LIN {X 0,Y 688.052,Z 1286.33,A -85,B 0,C 180,E1 33039.113,E2 33039.113} C_VEL
LIN {X 0,Y 687.976,Z 1293.841,A -85,B 0,C 180,E1 33037.347,E2 33037.347} C_VEL
LIN {X 0,Y 687.922,Z 1299.397,A -85,B 0,C 180,E1 33035.671,E2 33035.671} C_VEL
LIN {X 0,Y 687.911,Z 1303.97,A -85,B 0,C 180,E1 33033.749,E2 33033.749} C_VEL
LIN {X 0,Y 687.912,Z 1306.541,A -85,B 0,C 180,E1 33031.915,E2 33031.915} C_VEL
LIN {X 0,Y 687.913,Z 1307.484,A -85,B 0,C 180,E1 33030.082,E2 33030.082} C_VEL
LIN {X 0,Y 687.914,Z 1306.622,A -85,B 0,C 180,E1 33028.166,E2 33028.166} C_VEL
LIN {X 0,Y 687.914,Z 1304.122,A -85,B 0,C 180,E1 33026.332,E2 33026.332} C_VEL
LIN {X 0,Y 687.924,Z 1299.644,A -85,B 0,C 180,E1 33024.41,E2 33024.41} C_VEL
LIN {X 0,Y 687.974,Z 1294.146,A -85,B 0,C 180,E1 33022.735,E2 33022.735} C_VEL
LIN {X 0,Y 688.047,Z 1286.725,A -85,B 0,C 180,E1 33020.969,E2 33020.969} C_VEL
LIN {X 0,Y 688.172,Z 1277.229,A -85,B 0,C 180,E1 33019.176,E2 33019.176} C_VEL
LIN {X 0,Y 688.352,Z 1267.627,A -85,B 0,C 180,E1 33017.67,E2 33017.67} C_VEL
LIN {X 0,Y 688.626,Z 1255.593,A -85,B 0,C 180,E1 33016.052,E2 33016.052} C_VEL
LIN {X 0,Y 688.958,Z 1242.007,A -85,B 0,C 180,E1 33014.509,E2 33014.509} C_VEL
LIN {X 0,Y 689.355,Z 1227.995,A -85,B 0,C 180,E1 33013.136,E2 33013.136} C_VEL
LIN {X 0,Y 689.893,Z 1210.597,A -85,B 0,C 180,E1 33011.668,E2 33011.668} C_VEL
LIN {X 0,Y 690.479,Z 1192.469,A -85,B 0,C 180,E1 33010.368,E2 33010.368} C_VEL
LIN {X 0,Y 691.054,Z 1173.913,A -85,B 0,C 180,E1 33009.237,E2 33009.237} C_VEL
LIN {X 0,Y 691.686,Z 1153.527,A -85,B 0,C 180,E1 33008.19,E2 33008.19} C_VEL
LIN {X 0,Y 692.271,Z 1132.946,A -85,B 0,C 180,E1 33007.315,E2 33007.315} C_VEL
LIN {X 0,Y 692.788,Z 1111.812,A -85,B 0,C 180,E1 33006.587,E2 33006.587} C_VEL
LIN {X 0,Y 693.277,Z 1089.541,A -85,B 0,C 180,E1 33005.995,E2 33005.995} C_VEL
LIN {X 0,Y 693.611,Z 1067.293,A -85,B 0,C 180,E1 33005.565,E2 33005.565} C_VEL
LIN {X 0,Y 693.882,Z 1034.911,A -85,B 0,C 180,E1 33005.171,E2 33005.171} C_VEL
LIN {X 0,Y 694.12,Z 1007.188,A -85,B 0,C 180,E1 33004.852,E2 33004.852} C_VEL
LIN {X 0,Y 696.375,Z 998.353,A -85,B 0,C 180,E1 33004.529,E2 33004.529} C_VEL
LIN {X 0,Y 699.809,Z 987.003,A -85,B 0,C 180,E1 33004.278,E2 33004.278} C_VEL
LIN {X 0,Y 700.607,Z 984.081,A -85,B 0,C 180,E1 33004.196,E2 33004.196} C_VEL
LIN {X 0,Y 703.226,Z 974.14,A -85,B 0,C 180,E1 33003.891,E2 33003.891} C_VEL
LIN {X 0,Y 707.415,Z 958.39,A -85,B 0,C 180,E1 33003.611,E2 33003.611} C_VEL
LIN {X 0,Y 711.232,Z 939.749,A -85,B 0,C 180,E1 33003.422,E2 33003.422} C_VEL
LIN {X 0,Y 713.381,Z 919.951,A -85,B 0,C 180,E1 33003.244,E2 33003.244} C_VEL
LIN {X 0,Y 716.131,Z 876.116,A -85,B 0,C 180,E1 33002.811,E2 33002.811} C_VEL
LIN {X 0,Y 717.751,Z 866.34,A -85,B 0,C 180,E1 33002.56,E2 33002.56} C_VEL
LIN {X 0,Y 720.347,Z 841.246,A -85,B 0,C 180,E1 33002.165,E2 33002.165} C_VEL
LIN {X 0,Y 724.376,Z 790.008,A -85,B 0,C 180,E1 33001.568,E2 33001.568} C_VEL
LIN {X 0,Y 725.039,Z 781.425,A -85,B 0,C 180,E1 33001.471,E2 33001.471} C_VEL
LIN {X 0,Y 727.199,Z 793.678,A -85,B 0,C 180,E1 33001.159,E2 33001.159} C_VEL
LIN {X 0,Y 730.142,Z 804.778,A -85,B 0,C 180,E1 33000.743,E2 33000.743} C_VEL
LIN {X 0,Y 733.96,Z 814.871,A -85,B 0,C 180,E1 33000.215,E2 33000.215} C_VEL
LIN {X 0,Y 738.534,Z 823.545,A -85,B 0,C 180,E1 32999.601,E2 32999.601} C_VEL
LIN {X 0,Y 740.672,Z 827.583,A -85,B 0,C 180,E1 32999.211,E2 32999.211} C_VEL
LIN {X 0,Y 741.307,Z 830.76,A -85,B 0,C 180,E1 32998.777,E2 32998.777} C_VEL
LIN {X 0,Y 740.425,Z 833.197,A -85,B 0,C 180,E1 32998.296,E2 32998.296} C_VEL
LIN {X 0,Y 738.218,Z 834.451,A -85,B 0,C 180,E1 32997.838,E2 32997.838} C_VEL
LIN {X 0,Y 734.644,Z 834.531,A -85,B 0,C 180,E1 32997.385,E2 32997.385} C_VEL
LIN {X 0,Y 730.605,Z 833.461,A -85,B 0,C 180,E1 32997.029,E2 32997.029} C_VEL
LIN {X 0,Y 722.325,Z 829.141,A -85,B 0,C 180,E1 32996.443,E2 32996.443} C_VEL
LIN {X 0,Y 715.279,Z 823.545,A -85,B 0,C 180,E1 32995.849,E2 32995.849} C_VEL
LIN {X 0,Y 709.495,Z 816.874,A -85,B 0,C 180,E1 32995.248,E2 32995.248} C_VEL
LIN {X 0,Y 704.432,Z 808.219,A -85,B 0,C 180,E1 32994.563,E2 32994.563} C_VEL
LIN {X 0,Y 700.551,Z 797.694,A -85,B 0,C 180,E1 32993.817,E2 32993.817} C_VEL
LIN {X 0,Y 697.983,Z 785.051,A -85,B 0,C 180,E1 32993.01,E2 32993.01} C_VEL
LIN {X 0,Y 696.676,Z 766.868,A -85,B 0,C 180,E1 32991.949,E2 32991.949} C_VEL
LIN {X 0,Y 698.246,Z 704.476,A -85,B 0,C 180,E1 32988.524,E2 32988.524} C_VEL
LIN {X 0,Y 699.163,Z 671.327,A -85,B 0,C 180,E1 32986.649,E2 32986.649} C_VEL
LIN {X 0,Y 689.472,Z 649.922,A -85,B 0,C 180,E1 32984.698,E2 32984.698} C_VEL
LIN {X 0,Y 688.454,Z 646.906,A -85,B 0,C 180,E1 32984.431,E2 32984.431} C_VEL
LIN {X 0,Y 688.446,Z 646.914,A -85,B 0,C 180,E1 32981.458,E2 32981.458} C_VEL
LIN {X 0,Y 688.453,Z 646.914,A -85,B 0,C 180,E1 32978.479,E2 32978.479} C_VEL
LIN {X 0,Y 688.465,Z 646.915,A -85,B 0,C 180,E1 32975.435,E2 32975.435} C_VEL
LIN {X 0,Y 688.476,Z 647.124,A -85,B 0,C 180,E1 32972.456,E2 32972.456} C_VEL
LIN {X 0,Y 693.195,Z 663.428,A -85,B 0,C 180,E1 32970.946,E2 32970.946} C_VEL
LIN {X 0,Y 692.593,Z 691.38,A -85,B 0,C 180,E1 32968.687,E2 32968.687} C_VEL
LIN {X 0,Y 692.429,Z 700.611,A -85,B 0,C 180,E1 32967.953,E2 32967.953} C_VEL
LIN {X 0,Y 695.311,Z 714.317,A -85,B 0,C 180,E1 32967.669,E2 32967.669} C_VEL
LIN {X 0,Y 693.776,Z 994.51,A -85,B 0,C 180,E1 32964.567,E2 32964.567} C_VEL
LIN {X 0,Y 693.492,Z 1016.407,A -85,B 0,C 180,E1 32964.232,E2 32964.232} C_VEL
LIN {X 0,Y 693.064,Z 1038.792,A -85,B 0,C 180,E1 32963.733,E2 32963.733} C_VEL
LIN {X 0,Y 692.622,Z 1059.513,A -85,B 0,C 180,E1 32963.121,E2 32963.121} C_VEL
LIN {X 0,Y 692.072,Z 1079.43,A -85,B 0,C 180,E1 32962.383,E2 32962.383} C_VEL
LIN {X 0,Y 691.52,Z 1098.933,A -85,B 0,C 180,E1 32961.503,E2 32961.503} C_VEL
LIN {X 0,Y 690.941,Z 1117.723,A -85,B 0,C 180,E1 32960.5,E2 32960.5} C_VEL
LIN {X 0,Y 690.349,Z 1136.287,A -85,B 0,C 180,E1 32959.331,E2 32959.331} C_VEL
LIN {X 0,Y 689.813,Z 1153.31,A -85,B 0,C 180,E1 32958.071,E2 32958.071} C_VEL
LIN {X 0,Y 689.325,Z 1169.406,A -85,B 0,C 180,E1 32956.691,E2 32956.691} C_VEL
LIN {X 0,Y 688.911,Z 1184.069,A -85,B 0,C 180,E1 32955.231,E2 32955.231} C_VEL
LIN {X 0,Y 688.574,Z 1197.285,A -85,B 0,C 180,E1 32953.692,E2 32953.692} C_VEL
LIN {X 0,Y 688.318,Z 1209.092,A -85,B 0,C 180,E1 32952.075,E2 32952.075} C_VEL
LIN {X 0,Y 688.136,Z 1219.976,A -85,B 0,C 180,E1 32950.296,E2 32950.296} C_VEL
LIN {X 0,Y 688.015,Z 1228.491,A -85,B 0,C 180,E1 32948.609,E2 32948.609} C_VEL
LIN {X 0,Y 687.957,Z 1235.51,A -85,B 0,C 180,E1 32946.845,E2 32946.845} C_VEL
LIN {X 0,Y 687.914,Z 1241.082,A -85,B 0,C 180,E1 32945.003,E2 32945.003} C_VEL
LIN {X 0,Y 687.904,Z 1244.799,A -85,B 0,C 180,E1 32943.25,E2 32943.25} C_VEL
LIN {X 0,Y 687.909,Z 1246.913,A -85,B 0,C 180,E1 32941.416,E2 32941.416} C_VEL
LIN {X 0,Y 687.917,Z 1247.386,A -85,B 0,C 180,E1 32939.5,E2 32939.5} C_VEL
LIN {X 0,Y 687.906,Z 1246.182,A -85,B 0,C 180,E1 32937.667,E2 32937.667} C_VEL
LIN {X 0,Y 687.903,Z 1243.392,A -85,B 0,C 180,E1 32935.916,E2 32935.916} C_VEL
LIN {X 0,Y 687.927,Z 1238.788,A -85,B 0,C 180,E1 32934.077,E2 32934.077} C_VEL
LIN {X 0,Y 687.972,Z 1232.769,A -85,B 0,C 180,E1 32932.316,E2 32932.316} C_VEL
LIN {X 0,Y 688.058,Z 1224.885,A -85,B 0,C 180,E1 32930.548,E2 32930.548} C_VEL
LIN {X 0,Y 688.219,Z 1215.089,A -85,B 0,C 180,E1 32928.774,E2 32928.774} C_VEL
LIN {X 0,Y 688.427,Z 1203.628,A -85,B 0,C 180,E1 32927.054,E2 32927.054} C_VEL
LIN {X 0,Y 688.733,Z 1191.01,A -85,B 0,C 180,E1 32925.454,E2 32925.454} C_VEL
LIN {X 0,Y 689.115,Z 1176.622,A -85,B 0,C 180,E1 32923.911,E2 32923.911} C_VEL
LIN {X 0,Y 689.566,Z 1161.193,A -85,B 0,C 180,E1 32922.489,E2 32922.489} C_VEL
LIN {X 0,Y 690.092,Z 1144.286,A -85,B 0,C 180,E1 32921.149,E2 32921.149} C_VEL
LIN {X 0,Y 690.664,Z 1126.45,A -85,B 0,C 180,E1 32919.933,E2 32919.933} C_VEL
LIN {X 0,Y 691.261,Z 1107.52,A -85,B 0,C 180,E1 32918.845,E2 32918.845} C_VEL
LIN {X 0,Y 691.847,Z 1087.678,A -85,B 0,C 180,E1 32917.882,E2 32917.882} C_VEL
LIN {X 0,Y 692.178,Z 1075.526,A -85,B 0,C 180,E1 32917.373,E2 32917.373} C_VEL
LIN {X 0,Y 691.49,Z 1068.665,A -85,B 0,C 180,E1 32917.076,E2 32917.076} C_VEL
LIN {X 0,Y 686.397,Z 1051.614,A -85,B 0,C 180,E1 32916.295,E2 32916.295} C_VEL
LIN {X 0,Y 685.615,Z 1044.451,A -85,B 0,C 180,E1 32916.058,E2 32916.058} C_VEL
LIN {X 0,Y 686.063,Z 1022.443,A -85,B 0,C 180,E1 32915.52,E2 32915.52} C_VEL
LIN {X 0,Y 686.423,Z 1000.492,A -85,B 0,C 180,E1 32915.146,E2 32915.146} C_VEL
LIN {X 0,Y 688.095,Z 732.537,A -85,B 0,C 180,E1 32912.14,E2 32912.14} C_VEL
LIN {X 0,Y 687.988,Z 713.74,A -85,B 0,C 180,E1 32911.919,E2 32911.919} C_VEL
LIN {X 0,Y 684.931,Z 700.129,A -85,B 0,C 180,E1 32911.605,E2 32911.605} C_VEL
LIN {X 0,Y 685.853,Z 667.016,A -85,B 0,C 180,E1 32908.881,E2 32908.881} C_VEL
LIN {X 0,Y 685.402,Z 664.065,A -85,B 0,C 180,E1 32908.614,E2 32908.614} C_VEL
LIN {X 0,Y 680.514,Z 647.904,A -85,B 0,C 180,E1 32906.992,E2 32906.992} C_VEL
LIN {X 0,Y 680.521,Z 647.902,A -85,B 0,C 180,E1 32903.9,E2 32903.9} C_VEL
LIN {X 0,Y 680.516,Z 647.9,A -85,B 0,C 180,E1 32900.816,E2 32900.816} C_VEL
LIN {X 0,Y 680.522,Z 647.897,A -85,B 0,C 180,E1 32897.777,E2 32897.777} C_VEL
LIN {X 0,Y 680.52,Z 647.9,A -85,B 0,C 180,E1 32894.615,E2 32894.615} C_VEL
LIN {X 0,Y 680.53,Z 647.902,A -85,B 0,C 180,E1 32891.503,E2 32891.503} C_VEL
LIN {X 0,Y 680.525,Z 647.898,A -85,B 0,C 180,E1 32888.427,E2 32888.427} C_VEL
LIN {X 0,Y 680.52,Z 647.896,A -85,B 0,C 180,E1 32885.271,E2 32885.271} C_VEL
LIN {X 0,Y 680.519,Z 647.898,A -85,B 0,C 180,E1 32882.134,E2 32882.134} C_VEL
LIN {X 0,Y 680.531,Z 647.902,A -85,B 0,C 180,E1 32879.046,E2 32879.046} C_VEL
LIN {X 0,Y 680.521,Z 647.896,A -85,B 0,C 180,E1 32875.945,E2 32875.945} C_VEL
LIN {X 0,Y 680.524,Z 647.895,A -85,B 0,C 180,E1 32872.824,E2 32872.824} C_VEL
LIN {X 0,Y 680.52,Z 647.897,A -85,B 0,C 180,E1 32869.663,E2 32869.663} C_VEL
LIN {X 0,Y 680.525,Z 647.902,A -85,B 0,C 180,E1 32866.562,E2 32866.562} C_VEL
LIN {X 0,Y 680.523,Z 647.894,A -85,B 0,C 180,E1 32863.511,E2 32863.511} C_VEL
LIN {X 0,Y 680.521,Z 647.895,A -85,B 0,C 180,E1 32860.327,E2 32860.327} C_VEL
LIN {X 0,Y 680.521,Z 647.898,A -85,B 0,C 180,E1 32857.175,E2 32857.175} C_VEL
LIN {X 0,Y 680.522,Z 647.901,A -85,B 0,C 180,E1 32854.13,E2 32854.13} C_VEL
LIN {X 0,Y 680.524,Z 647.896,A -85,B 0,C 180,E1 32851.011,E2 32851.011} C_VEL
LIN {X 0,Y 680.523,Z 647.895,A -85,B 0,C 180,E1 32847.896,E2 32847.896} C_VEL
LIN {X 0,Y 680.522,Z 647.899,A -85,B 0,C 180,E1 32844.775,E2 32844.775} C_VEL
LIN {X 0,Y 680.525,Z 647.899,A -85,B 0,C 180,E1 32841.722,E2 32841.722} C_VEL
LIN {X 0,Y 680.522,Z 647.894,A -85,B 0,C 180,E1 32838.561,E2 32838.561} C_VEL
LIN {X 0,Y 680.524,Z 647.893,A -85,B 0,C 180,E1 32835.363,E2 32835.363} C_VEL
LIN {X 0,Y 680.52,Z 647.898,A -85,B 0,C 180,E1 32832.197,E2 32832.197} C_VEL
LIN {X 0,Y 680.524,Z 647.903,A -85,B 0,C 180,E1 32829.083,E2 32829.083} C_VEL
LIN {X 0,Y 680.524,Z 647.897,A -85,B 0,C 180,E1 32826.051,E2 32826.051} C_VEL
LIN {X 0,Y 680.526,Z 647.894,A -85,B 0,C 180,E1 32822.906,E2 32822.906} C_VEL
LIN {X 0,Y 680.522,Z 647.898,A -85,B 0,C 180,E1 32819.739,E2 32819.739} C_VEL
LIN {X 0,Y 680.524,Z 647.899,A -85,B 0,C 180,E1 32816.668,E2 32816.668} C_VEL
LIN {X 0,Y 680.521,Z 647.894,A -85,B 0,C 180,E1 32813.589,E2 32813.589} C_VEL
LIN {X 0,Y 680.528,Z 647.895,A -85,B 0,C 180,E1 32810.478,E2 32810.478} C_VEL
LIN {X 0,Y 680.518,Z 647.901,A -85,B 0,C 180,E1 32807.278,E2 32807.278} C_VEL
LIN {X 0,Y 680.525,Z 647.902,A -85,B 0,C 180,E1 32804.194,E2 32804.194} C_VEL
LIN {X 0,Y 680.516,Z 647.983,A -85,B 0,C 180,E1 32801.533,E2 32801.533} C_VEL
LIN {X 0,Y 687.339,Z 668.46,A -85,B 0,C 180,E1 32799.641,E2 32799.641} C_VEL
LIN {X 0,Y 686.324,Z 710.17,A -85,B 0,C 180,E1 32796.678,E2 32796.678} C_VEL
LIN {X 0,Y 685.036,Z 755.985,A -85,B 0,C 180,E1 32793.486,E2 32793.486} C_VEL
LIN {X 0,Y 683.854,Z 801.811,A -85,B 0,C 180,E1 32790.343,E2 32790.343} C_VEL
LIN {X 0,Y 682.807,Z 848.451,A -85,B 0,C 180,E1 32787.187,E2 32787.187} C_VEL
LIN {X 0,Y 681.979,Z 893.847,A -85,B 0,C 180,E1 32784.163,E2 32784.163} C_VEL
LIN {X 0,Y 682.461,Z 901.344,A -85,B 0,C 180,E1 32784.057,E2 32784.057} C_VEL
LIN {X 0,Y 681.831,Z 1024.236,A -85,B 0,C 180,E1 32782.694,E2 32782.694} C_VEL
LIN {X 0,Y 681.705,Z 1043.086,A -85,B 0,C 180,E1 32782.409,E2 32782.409} C_VEL
LIN {X 0,Y 681.562,Z 1057.156,A -85,B 0,C 180,E1 32782.059,E2 32782.059} C_VEL
LIN {X 0,Y 681.374,Z 1070.311,A -85,B 0,C 180,E1 32781.613,E2 32781.613} C_VEL
LIN {X 0,Y 681.169,Z 1082.604,A -85,B 0,C 180,E1 32781.078,E2 32781.078} C_VEL
LIN {X 0,Y 680.956,Z 1094.166,A -85,B 0,C 180,E1 32780.455,E2 32780.455} C_VEL
LIN {X 0,Y 680.77,Z 1105.02,A -85,B 0,C 180,E1 32779.744,E2 32779.744} C_VEL
LIN {X 0,Y 680.576,Z 1115.127,A -85,B 0,C 180,E1 32778.947,E2 32778.947} C_VEL
LIN {X 0,Y 680.397,Z 1124.558,A -85,B 0,C 180,E1 32778.052,E2 32778.052} C_VEL
LIN {X 0,Y 680.233,Z 1133.602,A -85,B 0,C 180,E1 32777.009,E2 32777.009} C_VEL
LIN {X 0,Y 680.099,Z 1142.811,A -85,B 0,C 180,E1 32775.645,E2 32775.645} C_VEL
LIN {X 0,Y 680.029,Z 1148.744,A -85,B 0,C 180,E1 32774.475,E2 32774.475} C_VEL
LIN {X 0,Y 679.997,Z 1153.042,A -85,B 0,C 180,E1 32773.348,E2 32773.348} C_VEL
LIN {X 0,Y 679.98,Z 1156.037,A -85,B 0,C 180,E1 32772.225,E2 32772.225} C_VEL
LIN {X 0,Y 679.976,Z 1157.82,A -85,B 0,C 180,E1 32771.107,E2 32771.107} C_VEL
LIN {X 0,Y 679.976,Z 1158.446,A -85,B 0,C 180,E1 32769.992,E2 32769.992} C_VEL
LIN {X 0,Y 679.98,Z 1157.896,A -85,B 0,C 180,E1 32768.841,E2 32768.841} C_VEL
LIN {X 0,Y 679.989,Z 1156.299,A -85,B 0,C 180,E1 32767.775,E2 32767.775} C_VEL
LIN {X 0,Y 680.009,Z 1153.501,A -85,B 0,C 180,E1 32766.671,E2 32766.671} C_VEL
LIN {X 0,Y 680.043,Z 1149.483,A -85,B 0,C 180,E1 32765.569,E2 32765.569} C_VEL
LIN {X 0,Y 680.109,Z 1144.147,A -85,B 0,C 180,E1 32764.469,E2 32764.469} C_VEL
LIN {X 0,Y 680.215,Z 1137.348,A -85,B 0,C 180,E1 32763.371,E2 32763.371} C_VEL
LIN {X 0,Y 680.395,Z 1128.078,A -85,B 0,C 180,E1 32762.185,E2 32762.185} C_VEL
LIN {X 0,Y 680.619,Z 1117.182,A -85,B 0,C 180,E1 32761.094,E2 32761.094} C_VEL
LIN {X 0,Y 680.839,Z 1106.279,A -85,B 0,C 180,E1 32760.21,E2 32760.21} C_VEL
LIN {X 0,Y 681.041,Z 1095.617,A -85,B 0,C 180,E1 32759.495,E2 32759.495} C_VEL
LIN {X 0,Y 681.246,Z 1084.216,A -85,B 0,C 180,E1 32758.865,E2 32758.865} C_VEL
LIN {X 0,Y 681.48,Z 1071.988,A -85,B 0,C 180,E1 32758.318,E2 32758.318} C_VEL
LIN {X 0,Y 681.666,Z 1058.753,A -85,B 0,C 180,E1 32757.856,E2 32757.856} C_VEL
LIN {X 0,Y 681.814,Z 1044.156,A -85,B 0,C 180,E1 32757.484,E2 32757.484} C_VEL
LIN {X 0,Y 681.926,Z 1026.393,A -85,B 0,C 180,E1 32757.206,E2 32757.206} C_VEL
LIN {X 0,Y 682.494,Z 951.65,A -85,B 0,C 180,E1 32756.322,E2 32756.322} C_VEL
LIN {X 0,Y 682.806,Z 896.544,A -85,B 0,C 180,E1 32755.66,E2 32755.66} C_VEL
LIN {X 0,Y 682.86,Z 890.86,A -85,B 0,C 180,E1 32755.296,E2 32755.296} C_VEL
LIN {X 0,Y 684.314,Z 844.923,A -85,B 0,C 180,E1 32752.106,E2 32752.106} C_VEL
LIN {X 0,Y 686.061,Z 799.923,A -85,B 0,C 180,E1 32748.908,E2 32748.908} C_VEL
LIN {X 0,Y 688.301,Z 755.929,A -85,B 0,C 180,E1 32745.702,E2 32745.702} C_VEL
LIN {X 0,Y 690.915,Z 714.185,A -85,B 0,C 180,E1 32742.568,E2 32742.568} C_VEL
LIN {X 0,Y 692.798,Z 677.036,A -85,B 0,C 180,E1 32739.601,E2 32739.601} C_VEL
LIN {X 0,Y 687.372,Z 663.531,A -85,B 0,C 180,E1 32737.908,E2 32737.908} C_VEL
LIN {X 0,Y 683.533,Z 655.104,A -85,B 0,C 180,E1 32736.725,E2 32736.725} C_VEL
LIN {X 0,Y 682.014,Z 651.668,A -85,B 0,C 180,E1 32736.223,E2 32736.223} C_VEL
LIN {X 0,Y 680.706,Z 648.913,A -85,B 0,C 180,E1 32735.804,E2 32735.804} C_VEL
LIN {X 0,Y 680.52,Z 647.9,A -85,B 0,C 180,E1 32735.671,E2 32735.671} C_VEL
LIN {X 0,Y 680.52,Z 647.902,A -85,B 0,C 180,E1 32732.525,E2 32732.525} C_VEL
LIN {X 0,Y 680.526,Z 647.898,A -85,B 0,C 180,E1 32729.346,E2 32729.346} C_VEL
LIN {X 0,Y 680.522,Z 647.904,A -85,B 0,C 180,E1 32726.161,E2 32726.161} C_VEL
LIN {X 0,Y 680.524,Z 647.898,A -85,B 0,C 180,E1 32723.06,E2 32723.06} C_VEL
LIN {X 0,Y 680.527,Z 647.901,A -85,B 0,C 180,E1 32719.943,E2 32719.943} C_VEL
LIN {X 0,Y 680.523,Z 647.9,A -85,B 0,C 180,E1 32716.781,E2 32716.781} C_VEL
LIN {X 0,Y 680.537,Z 648.001,A -85,B 0,C 180,E1 32715.741,E2 32715.741} C_VEL
LIN {X 0,Y 681.774,Z 651.333,A -85,B 0,C 180,E1 32715.372,E2 32715.372} C_VEL
LIN {X 0,Y 682.888,Z 653.487,A -85,B 0,C 180,E1 32715.11,E2 32715.11} C_VEL
LIN {X 0,Y 687.786,Z 664.015,A -85,B 0,C 180,E1 32713.976,E2 32713.976} C_VEL
LIN {X 0,Y 691.216,Z 672.497,A -85,B 0,C 180,E1 32713.172,E2 32713.172} C_VEL
LIN {X 0,Y 688.619,Z 719.746,A -85,B 0,C 180,E1 32710.523,E2 32710.523} C_VEL
LIN {X 0,Y 687.369,Z 766.196,A -85,B 0,C 180,E1 32708.026,E2 32708.026} C_VEL
LIN {X 0,Y 688.944,Z 785.514,A -85,B 0,C 180,E1 32706.929,E2 32706.929} C_VEL
LIN {X 0,Y 692.056,Z 799.714,A -85,B 0,C 180,E1 32706.062,E2 32706.062} C_VEL
LIN {X 0,Y 696.525,Z 811.165,A -85,B 0,C 180,E1 32705.303,E2 32705.303} C_VEL
LIN {X 0,Y 702.239,Z 820.654,A -85,B 0,C 180,E1 32704.614,E2 32704.614} C_VEL
LIN {X 0,Y 709.083,Z 828.478,A -85,B 0,C 180,E1 32703.988,E2 32703.988} C_VEL
LIN {X 0,Y 717.318,Z 835.074,A -85,B 0,C 180,E1 32703.388,E2 32703.388} C_VEL
LIN {X 0,Y 726.337,Z 840.033,A -85,B 0,C 180,E1 32702.844,E2 32702.844} C_VEL
LIN {X 0,Y 731.268,Z 841.551,A -85,B 0,C 180,E1 32702.472,E2 32702.472} C_VEL
LIN {X 0,Y 735.317,Z 841.711,A -85,B 0,C 180,E1 32702.026,E2 32702.026} C_VEL
LIN {X 0,Y 738.021,Z 840.588,A -85,B 0,C 180,E1 32701.549,E2 32701.549} C_VEL
LIN {X 0,Y 739.249,Z 838.373,A -85,B 0,C 180,E1 32701.068,E2 32701.068} C_VEL
LIN {X 0,Y 738.904,Z 835.208,A -85,B 0,C 180,E1 32700.603,E2 32700.603} C_VEL
LIN {X 0,Y 737.005,Z 831.347,A -85,B 0,C 180,E1 32700.197,E2 32700.197} C_VEL
LIN {X 0,Y 732.153,Z 822.678,A -85,B 0,C 180,E1 32699.537,E2 32699.537} C_VEL
LIN {X 0,Y 728.061,Z 812.657,A -85,B 0,C 180,E1 32698.964,E2 32698.964} C_VEL
LIN {X 0,Y 726.84,Z 809.083,A -85,B 0,C 180,E1 32698.789,E2 32698.789} C_VEL
LIN {X 0,Y 723.154,Z 852.196,A -85,B 0,C 180,E1 32698.253,E2 32698.253} C_VEL
LIN {X 0,Y 720.83,Z 872.102,A -85,B 0,C 180,E1 32697.907,E2 32697.907} C_VEL
LIN {X 0,Y 719.496,Z 880.295,A -85,B 0,C 180,E1 32697.706,E2 32697.706} C_VEL
LIN {X 0,Y 717.196,Z 912.709,A -85,B 0,C 180,E1 32697.417,E2 32697.417} C_VEL
LIN {X 0,Y 713.888,Z 932.091,A -85,B 0,C 180,E1 32697.277,E2 32697.277} C_VEL
LIN {X 0,Y 708.832,Z 950.724,A -85,B 0,C 180,E1 32697.129,E2 32697.129} C_VEL
LIN {X 0,Y 703.102,Z 967.543,A -85,B 0,C 180,E1 32696.885,E2 32696.885} C_VEL
LIN {X 0,Y 698.713,Z 980.481,A -85,B 0,C 180,E1 32696.567,E2 32696.567} C_VEL
LIN {X 0,Y 696.39,Z 988.262,A -85,B 0,C 180,E1 32696.311,E2 32696.311} C_VEL
LIN {X 0,Y 691.992,Z 1000.207,A -85,B 0,C 180,E1 32696.004,E2 32696.004} C_VEL
LIN {X 0,Y 686.96,Z 1018.232,A -85,B 0,C 180,E1 32695.334,E2 32695.334} C_VEL
LIN {X 0,Y 686.704,Z 1020.499,A -85,B 0,C 180,E1 32695.269,E2 32695.269} C_VEL
LIN {X 0,Y 686.367,Z 1064.962,A -85,B 0,C 180,E1 32694.747,E2 32694.747} C_VEL
LIN {X 0,Y 685.968,Z 1087.624,A -85,B 0,C 180,E1 32694.321,E2 32694.321} C_VEL
LIN {X 0,Y 685.459,Z 1109.858,A -85,B 0,C 180,E1 32693.74,E2 32693.74} C_VEL
LIN {X 0,Y 684.902,Z 1130.772,A -85,B 0,C 180,E1 32693.031,E2 32693.031} C_VEL
LIN {X 0,Y 684.264,Z 1150.713,A -85,B 0,C 180,E1 32692.196,E2 32692.196} C_VEL
LIN {X 0,Y 683.586,Z 1170.799,A -85,B 0,C 180,E1 32691.178,E2 32691.178} C_VEL
LIN {X 0,Y 682.88,Z 1190.505,A -85,B 0,C 180,E1 32689.991,E2 32689.991} C_VEL
LIN {X 0,Y 682.27,Z 1207.173,A -85,B 0,C 180,E1 32688.808,E2 32688.808} C_VEL
LIN {X 0,Y 681.752,Z 1222.321,A -85,B 0,C 180,E1 32687.574,E2 32687.574} C_VEL
LIN {X 0,Y 681.21,Z 1238.743,A -85,B 0,C 180,E1 32686.017,E2 32686.017} C_VEL
LIN {X 0,Y 680.808,Z 1252.024,A -85,B 0,C 180,E1 32684.544,E2 32684.544} C_VEL
LIN {X 0,Y 680.488,Z 1264.752,A -85,B 0,C 180,E1 32682.904,E2 32682.904} C_VEL
LIN {X 0,Y 680.245,Z 1275.334,A -85,B 0,C 180,E1 32681.272,E2 32681.272} C_VEL
LIN {X 0,Y 680.099,Z 1284.685,A -85,B 0,C 180,E1 32679.562,E2 32679.562} C_VEL
LIN {X 0,Y 679.983,Z 1293.042,A -85,B 0,C 180,E1 32677.65,E2 32677.65} C_VEL
LIN {X 0,Y 679.928,Z 1298.638,A -85,B 0,C 180,E1 32675.992,E2 32675.992} C_VEL
LIN {X 0,Y 679.918,Z 1303.173,A -85,B 0,C 180,E1 32674.216,E2 32674.216} C_VEL
LIN {X 0,Y 679.905,Z 1306.206,A -85,B 0,C 180,E1 32672.274,E2 32672.274} C_VEL
LIN {X 0,Y 679.899,Z 1307.374,A -85,B 0,C 180,E1 32670.504,E2 32670.504} C_VEL
LIN {X 0,Y 679.905,Z 1307.039,A -85,B 0,C 180,E1 32668.651,E2 32668.651} C_VEL
LIN {X 0,Y 679.918,Z 1304.96,A -85,B 0,C 180,E1 32666.795,E2 32666.795} C_VEL
LIN {X 0,Y 679.919,Z 1301.409,A -85,B 0,C 180,E1 32665.021,E2 32665.021} C_VEL
LIN {X 0,Y 679.954,Z 1295.529,A -85,B 0,C 180,E1 32663.031,E2 32663.031} C_VEL
LIN {X 0,Y 680.026,Z 1289.007,A -85,B 0,C 180,E1 32661.373,E2 32661.373} C_VEL
LIN {X 0,Y 680.147,Z 1280.704,A -85,B 0,C 180,E1 32659.667,E2 32659.667} C_VEL
LIN {X 0,Y 680.362,Z 1269.933,A -85,B 0,C 180,E1 32657.867,E2 32657.867} C_VEL
LIN {X 0,Y 680.599,Z 1259.582,A -85,B 0,C 180,E1 32656.404,E2 32656.404} C_VEL
LIN {X 0,Y 680.969,Z 1246.821,A -85,B 0,C 180,E1 32654.848,E2 32654.848} C_VEL
LIN {X 0,Y 681.437,Z 1231.675,A -85,B 0,C 180,E1 32653.285,E2 32653.285} C_VEL
LIN {X 0,Y 681.901,Z 1217.561,A -85,B 0,C 180,E1 32652.021,E2 32652.021} C_VEL
LIN {X 0,Y 682.55,Z 1199.679,A -85,B 0,C 180,E1 32650.634,E2 32650.634} C_VEL
LIN {X 0,Y 683.208,Z 1181.388,A -85,B 0,C 180,E1 32649.436,E2 32649.436} C_VEL
LIN {X 0,Y 683.913,Z 1161.279,A -85,B 0,C 180,E1 32648.317,E2 32648.317} C_VEL
LIN {X 0,Y 684.579,Z 1140.801,A -85,B 0,C 180,E1 32647.368,E2 32647.368} C_VEL
LIN {X 0,Y 685.204,Z 1120,A -85,B 0,C 180,E1 32646.584,E2 32646.584} C_VEL
LIN {X 0,Y 685.736,Z 1098.158,A -85,B 0,C 180,E1 32645.934,E2 32645.934} C_VEL
LIN {X 0,Y 686.201,Z 1075.524,A -85,B 0,C 180,E1 32645.43,E2 32645.43} C_VEL
LIN {X 0,Y 686.506,Z 1052.82,A -85,B 0,C 180,E1 32645.09,E2 32645.09} C_VEL
LIN {X 0,Y 686.72,Z 1019.378,A -85,B 0,C 180,E1 32644.716,E2 32644.716} C_VEL
LIN {X 0,Y 689.076,Z 1010.58,A -85,B 0,C 180,E1 32644.378,E2 32644.378} C_VEL
LIN {X 0,Y 692.385,Z 999.018,A -85,B 0,C 180,E1 32643.958,E2 32643.958} C_VEL
LIN {X 0,Y 697.031,Z 986.43,A -85,B 0,C 180,E1 32643.641,E2 32643.641} C_VEL
LIN {X 0,Y 700.117,Z 976.148,A -85,B 0,C 180,E1 32643.309,E2 32643.309} C_VEL
LIN {X 0,Y 705.431,Z 960.919,A -85,B 0,C 180,E1 32643.001,E2 32643.001} C_VEL
LIN {X 0,Y 711.215,Z 942.746,A -85,B 0,C 180,E1 32642.799,E2 32642.799} C_VEL
LIN {X 0,Y 715.636,Z 923.297,A -85,B 0,C 180,E1 32642.661,E2 32642.661} C_VEL
LIN {X 0,Y 718.054,Z 903.887,A -85,B 0,C 180,E1 32642.51,E2 32642.51} C_VEL
LIN {X 0,Y 719.734,Z 878.318,A -85,B 0,C 180,E1 32642.258,E2 32642.258} C_VEL
LIN {X 0,Y 721.546,Z 866.843,A -85,B 0,C 180,E1 32641.985,E2 32641.985} C_VEL
LIN {X 0,Y 724.354,Z 839.363,A -85,B 0,C 180,E1 32641.571,E2 32641.571} C_VEL
LIN {X 0,Y 726.867,Z 809.074,A -85,B 0,C 180,E1 32641.207,E2 32641.207} C_VEL
LIN {X 0,Y 730.815,Z 819.741,A -85,B 0,C 180,E1 32640.649,E2 32640.649} C_VEL
LIN {X 0,Y 735.518,Z 828.972,A -85,B 0,C 180,E1 32640.004,E2 32640.004} C_VEL
LIN {X 0,Y 738.401,Z 833.908,A -85,B 0,C 180,E1 32639.55,E2 32639.55} C_VEL
LIN {X 0,Y 739.315,Z 837.368,A -85,B 0,C 180,E1 32639.096,E2 32639.096} C_VEL
LIN {X 0,Y 738.731,Z 839.774,A -85,B 0,C 180,E1 32638.658,E2 32638.658} C_VEL
LIN {X 0,Y 736.661,Z 841.37,A -85,B 0,C 180,E1 32638.178,E2 32638.178} C_VEL
LIN {X 0,Y 733.239,Z 841.795,A -85,B 0,C 180,E1 32637.723,E2 32637.723} C_VEL
LIN {X 0,Y 729.146,Z 841.045,A -85,B 0,C 180,E1 32637.351,E2 32637.351} C_VEL
LIN {X 0,Y 720.717,Z 837.341,A -85,B 0,C 180,E1 32636.781,E2 32636.781} C_VEL
LIN {X 0,Y 711.983,Z 831.314,A -85,B 0,C 180,E1 32636.098,E2 32636.098} C_VEL
LIN {X 0,Y 704.692,Z 823.772,A -85,B 0,C 180,E1 32635.383,E2 32635.383} C_VEL
LIN {X 0,Y 698.872,Z 814.742,A -85,B 0,C 180,E1 32634.638,E2 32634.638} C_VEL
LIN {X 0,Y 694.538,Z 804.25,A -85,B 0,C 180,E1 32633.867,E2 32633.867} C_VEL
LIN {X 0,Y 691.369,Z 790.698,A -85,B 0,C 180,E1 32632.971,E2 32632.971} C_VEL
LIN {X 0,Y 689.792,Z 773.139,A -85,B 0,C 180,E1 32631.916,E2 32631.916} C_VEL
LIN {X 0,Y 690.364,Z 739.385,A -85,B 0,C 180,E1 32630.047,E2 32630.047} C_VEL
LIN {X 0,Y 692.118,Z 688.182,A -85,B 0,C 180,E1 32627.183,E2 32627.183} C_VEL
LIN {X 0,Y 692.384,Z 674.791,A -85,B 0,C 180,E1 32626.405,E2 32626.405} C_VEL
LIN {X 0,Y 681.944,Z 651.548,A -85,B 0,C 180,E1 32624.261,E2 32624.261} C_VEL
LIN {X 0,Y 680.519,Z 647.971,A -85,B 0,C 180,E1 32623.935,E2 32623.935} C_VEL
LIN {X 0,Y 680.531,Z 647.901,A -85,B 0,C 180,E1 32620.827,E2 32620.827} C_VEL
LIN {X 0,Y 680.514,Z 647.903,A -85,B 0,C 180,E1 32617.768,E2 32617.768} C_VEL
LIN {X 0,Y 680.523,Z 647.902,A -85,B 0,C 180,E1 32614.654,E2 32614.654} C_VEL
LIN {X 0,Y 680.529,Z 647.913,A -85,B 0,C 180,E1 32612.794,E2 32612.794} C_VEL
LIN {X 0,Y 685.809,Z 665.432,A -85,B 0,C 180,E1 32611.148,E2 32611.148} C_VEL
LIN {X 0,Y 685.166,Z 697.042,A -85,B 0,C 180,E1 32608.598,E2 32608.598} C_VEL
LIN {X 0,Y 685.16,Z 701.343,A -85,B 0,C 180,E1 32608.27,E2 32608.27} C_VEL
LIN {X 0,Y 688.184,Z 715.662,A -85,B 0,C 180,E1 32607.959,E2 32607.959} C_VEL
LIN {X 0,Y 686.505,Z 994.28,A -85,B 0,C 180,E1 32604.849,E2 32604.849} C_VEL
LIN {X 0,Y 686.186,Z 1016.266,A -85,B 0,C 180,E1 32604.509,E2 32604.509} C_VEL
LIN {X 0,Y 685.713,Z 1038.685,A -85,B 0,C 180,E1 32604.006,E2 32604.006} C_VEL
LIN {X 0,Y 685.217,Z 1059.551,A -85,B 0,C 180,E1 32603.385,E2 32603.385} C_VEL
LIN {X 0,Y 684.589,Z 1079.974,A -85,B 0,C 180,E1 32602.619,E2 32602.619} C_VEL
LIN {X 0,Y 683.956,Z 1099.827,A -85,B 0,C 180,E1 32601.707,E2 32601.707} C_VEL
LIN {X 0,Y 683.265,Z 1119.611,A -85,B 0,C 180,E1 32600.625,E2 32600.625} C_VEL
LIN {X 0,Y 682.626,Z 1137.637,A -85,B 0,C 180,E1 32599.465,E2 32599.465} C_VEL
LIN {X 0,Y 682.015,Z 1154.908,A -85,B 0,C 180,E1 32598.157,E2 32598.157} C_VEL
LIN {X 0,Y 681.485,Z 1170.326,A -85,B 0,C 180,E1 32596.801,E2 32596.801} C_VEL
LIN {X 0,Y 681,Z 1185.626,A -85,B 0,C 180,E1 32595.238,E2 32595.238} C_VEL
LIN {X 0,Y 680.635,Z 1198.669,A -85,B 0,C 180,E1 32593.681,E2 32593.681} C_VEL
LIN {X 0,Y 680.351,Z 1210.231,A -85,B 0,C 180,E1 32592.046,E2 32592.046} C_VEL
LIN {X 0,Y 680.153,Z 1220.898,A -85,B 0,C 180,E1 32590.246,E2 32590.246} C_VEL
LIN {X 0,Y 680.016,Z 1229.578,A -85,B 0,C 180,E1 32588.455,E2 32588.455} C_VEL
LIN {X 0,Y 679.957,Z 1236.113,A -85,B 0,C 180,E1 32586.756,E2 32586.756} C_VEL
LIN {X 0,Y 679.915,Z 1241.288,A -85,B 0,C 180,E1 32584.978,E2 32584.978} C_VEL
LIN {X 0,Y 679.902,Z 1244.934,A -85,B 0,C 180,E1 32583.204,E2 32583.204} C_VEL
LIN {X 0,Y 679.907,Z 1246.98,A -85,B 0,C 180,E1 32581.348,E2 32581.348} C_VEL
LIN {X 0,Y 679.917,Z 1247.385,A -85,B 0,C 180,E1 32579.494,E2 32579.494} C_VEL
LIN {X 0,Y 679.907,Z 1246.181,A -85,B 0,C 180,E1 32577.64,E2 32577.64} C_VEL
LIN {X 0,Y 679.905,Z 1243.39,A -85,B 0,C 180,E1 32575.868,E2 32575.868} C_VEL
LIN {X 0,Y 679.93,Z 1238.787,A -85,B 0,C 180,E1 32574.007,E2 32574.007} C_VEL
LIN {X 0,Y 679.986,Z 1232.766,A -85,B 0,C 180,E1 32572.225,E2 32572.225} C_VEL
LIN {X 0,Y 680.079,Z 1224.883,A -85,B 0,C 180,E1 32570.437,E2 32570.437} C_VEL
LIN {X 0,Y 680.263,Z 1215.085,A -85,B 0,C 180,E1 32568.641,E2 32568.641} C_VEL
LIN {X 0,Y 680.502,Z 1203.778,A -85,B 0,C 180,E1 32566.922,E2 32566.922} C_VEL
LIN {X 0,Y 680.85,Z 1191.005,A -85,B 0,C 180,E1 32565.282,E2 32565.282} C_VEL
LIN {X 0,Y 681.279,Z 1176.524,A -85,B 0,C 180,E1 32563.711,E2 32563.711} C_VEL
LIN {X 0,Y 681.801,Z 1160.682,A -85,B 0,C 180,E1 32562.239,E2 32562.239} C_VEL
LIN {X 0,Y 682.426,Z 1143.072,A -85,B 0,C 180,E1 32560.84,E2 32560.84} C_VEL
LIN {X 0,Y 683.049,Z 1125.807,A -85,B 0,C 180,E1 32559.661,E2 32559.661} C_VEL
LIN {X 0,Y 683.721,Z 1106.708,A -85,B 0,C 180,E1 32558.555,E2 32558.555} C_VEL
LIN {X 0,Y 684.348,Z 1087.806,A -85,B 0,C 180,E1 32557.633,E2 32557.633} C_VEL
LIN {X 0,Y 684.964,Z 1068.289,A -85,B 0,C 180,E1 32556.833,E2 32556.833} C_VEL
LIN {X 0,Y 685.543,Z 1047.136,A -85,B 0,C 180,E1 32556.136,E2 32556.136} C_VEL
LIN {X 0,Y 685.615,Z 1044.451,A -85,B 0,C 180,E1 32556.058,E2 32556.058} C_VEL
LIN {X 0,Y 684.898,Z 1037.193,A -85,B 0,C 180,E1 32555.832,E2 32555.832} C_VEL
LIN {X 0,Y 679.819,Z 1019.206,A -85,B 0,C 180,E1 32555.21,E2 32555.21} C_VEL
LIN {X 0,Y 678.959,Z 1011.799,A -85,B 0,C 180,E1 32555.038,E2 32555.038} C_VEL
LIN {X 0,Y 679.302,Z 986.275,A -85,B 0,C 180,E1 32554.686,E2 32554.686} C_VEL
LIN {X 0,Y 681.122,Z 716.142,A -85,B 0,C 180,E1 32551.64,E2 32551.64} C_VEL
LIN {X 0,Y 677.569,Z 700.346,A -85,B 0,C 180,E1 32551.268,E2 32551.268} C_VEL
LIN {X 0,Y 678.519,Z 668.383,A -85,B 0,C 180,E1 32548.622,E2 32548.622} C_VEL
LIN {X 0,Y 672.568,Z 648.893,A -85,B 0,C 180,E1 32546.65,E2 32546.65} C_VEL
LIN {X 0,Y 672.568,Z 648.891,A -85,B 0,C 180,E1 32543.686,E2 32543.686} C_VEL
LIN {X 0,Y 672.572,Z 648.892,A -85,B 0,C 180,E1 32540.704,E2 32540.704} C_VEL
LIN {X 0,Y 672.575,Z 648.887,A -85,B 0,C 180,E1 32537.636,E2 32537.636} C_VEL
LIN {X 0,Y 672.578,Z 648.888,A -85,B 0,C 180,E1 32534.564,E2 32534.564} C_VEL
LIN {X 0,Y 672.591,Z 648.892,A -85,B 0,C 180,E1 32531.473,E2 32531.473} C_VEL
LIN {X 0,Y 672.585,Z 648.887,A -85,B 0,C 180,E1 32528.42,E2 32528.42} C_VEL
LIN {X 0,Y 672.579,Z 648.885,A -85,B 0,C 180,E1 32525.228,E2 32525.228} C_VEL
LIN {X 0,Y 672.582,Z 648.887,A -85,B 0,C 180,E1 32522.156,E2 32522.156} C_VEL
LIN {X 0,Y 672.593,Z 648.89,A -85,B 0,C 180,E1 32519.057,E2 32519.057} C_VEL
LIN {X 0,Y 672.582,Z 648.886,A -85,B 0,C 180,E1 32515.917,E2 32515.917} C_VEL
LIN {X 0,Y 672.585,Z 648.884,A -85,B 0,C 180,E1 32512.821,E2 32512.821} C_VEL
LIN {X 0,Y 672.584,Z 648.886,A -85,B 0,C 180,E1 32509.723,E2 32509.723} C_VEL
LIN {X 0,Y 672.586,Z 648.89,A -85,B 0,C 180,E1 32506.675,E2 32506.675} C_VEL
LIN {X 0,Y 672.584,Z 648.883,A -85,B 0,C 180,E1 32503.498,E2 32503.498} C_VEL
LIN {X 0,Y 672.583,Z 648.884,A -85,B 0,C 180,E1 32500.364,E2 32500.364} C_VEL
LIN {X 0,Y 672.582,Z 648.886,A -85,B 0,C 180,E1 32497.175,E2 32497.175} C_VEL
LIN {X 0,Y 672.583,Z 648.889,A -85,B 0,C 180,E1 32494.093,E2 32494.093} C_VEL
LIN {X 0,Y 672.583,Z 648.886,A -85,B 0,C 180,E1 32490.938,E2 32490.938} C_VEL
LIN {X 0,Y 672.579,Z 648.884,A -85,B 0,C 180,E1 32487.786,E2 32487.786} C_VEL
LIN {X 0,Y 672.582,Z 648.887,A -85,B 0,C 180,E1 32484.713,E2 32484.713} C_VEL
LIN {X 0,Y 672.589,Z 648.889,A -85,B 0,C 180,E1 32481.624,E2 32481.624} C_VEL
LIN {X 0,Y 672.583,Z 648.883,A -85,B 0,C 180,E1 32478.511,E2 32478.511} C_VEL
LIN {X 0,Y 672.585,Z 648.882,A -85,B 0,C 180,E1 32475.362,E2 32475.362} C_VEL
LIN {X 0,Y 672.584,Z 648.887,A -85,B 0,C 180,E1 32472.258,E2 32472.258} C_VEL
LIN {X 0,Y 672.587,Z 648.89,A -85,B 0,C 180,E1 32469.189,E2 32469.189} C_VEL
LIN {X 0,Y 672.585,Z 648.886,A -85,B 0,C 180,E1 32466.057,E2 32466.057} C_VEL
LIN {X 0,Y 672.583,Z 648.883,A -85,B 0,C 180,E1 32462.847,E2 32462.847} C_VEL
LIN {X 0,Y 672.584,Z 648.888,A -85,B 0,C 180,E1 32459.739,E2 32459.739} C_VEL
LIN {X 0,Y 672.583,Z 648.889,A -85,B 0,C 180,E1 32456.631,E2 32456.631} C_VEL
LIN {X 0,Y 672.58,Z 648.884,A -85,B 0,C 180,E1 32453.514,E2 32453.514} C_VEL
LIN {X 0,Y 672.583,Z 648.885,A -85,B 0,C 180,E1 32450.362,E2 32450.362} C_VEL
LIN {X 0,Y 672.577,Z 648.89,A -85,B 0,C 180,E1 32447.206,E2 32447.206} C_VEL
LIN {X 0,Y 672.582,Z 648.891,A -85,B 0,C 180,E1 32444.087,E2 32444.087} C_VEL
LIN {X 0,Y 672.6,Z 649.071,A -85,B 0,C 180,E1 32441.914,E2 32441.914} C_VEL
LIN {X 0,Y 680.12,Z 671.368,A -85,B 0,C 180,E1 32439.817,E2 32439.817} C_VEL
LIN {X 0,Y 679.013,Z 712.379,A -85,B 0,C 180,E1 32436.88,E2 32436.88} C_VEL
LIN {X 0,Y 677.635,Z 758.034,A -85,B 0,C 180,E1 32433.677,E2 32433.677} C_VEL
LIN {X 0,Y 676.336,Z 804.308,A -85,B 0,C 180,E1 32430.473,E2 32430.473} C_VEL
LIN {X 0,Y 675.184,Z 851.827,A -85,B 0,C 180,E1 32427.233,E2 32427.233} C_VEL
LIN {X 0,Y 674.37,Z 894.68,A -85,B 0,C 180,E1 32424.369,E2 32424.369} C_VEL
LIN {X 0,Y 674.863,Z 901.834,A -85,B 0,C 180,E1 32424.266,E2 32424.266} C_VEL
LIN {X 0,Y 674.455,Z 961.662,A -85,B 0,C 180,E1 32423.584,E2 32423.584} C_VEL
LIN {X 0,Y 674.106,Z 1023.1,A -85,B 0,C 180,E1 32422.882,E2 32422.882} C_VEL
LIN {X 0,Y 673.967,Z 1043.319,A -85,B 0,C 180,E1 32422.581,E2 32422.581} C_VEL
LIN {X 0,Y 673.808,Z 1058.029,A -85,B 0,C 180,E1 32422.211,E2 32422.211} C_VEL
LIN {X 0,Y 673.598,Z 1071.679,A -85,B 0,C 180,E1 32421.738,E2 32421.738} C_VEL
LIN {X 0,Y 673.356,Z 1084.747,A -85,B 0,C 180,E1 32421.152,E2 32421.152} C_VEL
LIN {X 0,Y 673.11,Z 1097.548,A -85,B 0,C 180,E1 32420.432,E2 32420.432} C_VEL
LIN {X 0,Y 672.84,Z 1110.95,A -85,B 0,C 180,E1 32419.485,E2 32419.485} C_VEL
LIN {X 0,Y 672.597,Z 1122.428,A -85,B 0,C 180,E1 32418.46,E2 32418.46} C_VEL
LIN {X 0,Y 672.402,Z 1131.363,A -85,B 0,C 180,E1 32417.481,E2 32417.481} C_VEL
LIN {X 0,Y 672.254,Z 1139.285,A -85,B 0,C 180,E1 32416.416,E2 32416.416} C_VEL
LIN {X 0,Y 672.159,Z 1145.636,A -85,B 0,C 180,E1 32415.355,E2 32415.355} C_VEL
LIN {X 0,Y 672.09,Z 1150.996,A -85,B 0,C 180,E1 32414.21,E2 32414.21} C_VEL
LIN {X 0,Y 672.05,Z 1155.476,A -85,B 0,C 180,E1 32412.896,E2 32412.896} C_VEL
LIN {X 0,Y 672.035,Z 1158.551,A -85,B 0,C 180,E1 32411.345,E2 32411.345} C_VEL
LIN {X 0,Y 672.035,Z 1159.417,A -85,B 0,C 180,E1 32410.025,E2 32410.025} C_VEL
LIN {X 0,Y 672.043,Z 1158.869,A -85,B 0,C 180,E1 32408.815,E2 32408.815} C_VEL
LIN {X 0,Y 672.056,Z 1157.016,A -85,B 0,C 180,E1 32407.609,E2 32407.609} C_VEL
LIN {X 0,Y 672.09,Z 1153.561,A -85,B 0,C 180,E1 32406.321,E2 32406.321} C_VEL
LIN {X 0,Y 672.176,Z 1147.615,A -85,B 0,C 180,E1 32404.864,E2 32404.864} C_VEL
LIN {X 0,Y 672.304,Z 1140.329,A -85,B 0,C 180,E1 32403.581,E2 32403.581} C_VEL
LIN {X 0,Y 672.473,Z 1132.278,A -85,B 0,C 180,E1 32402.471,E2 32402.471} C_VEL
LIN {X 0,Y 672.692,Z 1123.114,A -85,B 0,C 180,E1 32401.448,E2 32401.448} C_VEL
LIN {X 0,Y 672.963,Z 1111.281,A -85,B 0,C 180,E1 32400.383,E2 32400.383} C_VEL
LIN {X 0,Y 673.247,Z 1098.811,A -85,B 0,C 180,E1 32399.489,E2 32399.489} C_VEL
LIN {X 0,Y 673.487,Z 1086.219,A -85,B 0,C 180,E1 32398.766,E2 32398.766} C_VEL
LIN {X 0,Y 673.755,Z 1073.219,A -85,B 0,C 180,E1 32398.172,E2 32398.172} C_VEL
LIN {X 0,Y 673.972,Z 1058.76,A -85,B 0,C 180,E1 32397.662,E2 32397.662} C_VEL
LIN {X 0,Y 674.13,Z 1043.142,A -85,B 0,C 180,E1 32397.272,E2 32397.272} C_VEL
LIN {X 0,Y 674.303,Z 1019.372,A -85,B 0,C 180,E1 32396.932,E2 32396.932} C_VEL
LIN {X 0,Y 675.37,Z 897.662,A -85,B 0,C 180,E1 32395.42,E2 32395.42} C_VEL
LIN {X 0,Y 676.725,Z 854.866,A -85,B 0,C 180,E1 32392.444,E2 32392.444} C_VEL
LIN {X 0,Y 678.73,Z 807.39,A -85,B 0,C 180,E1 32389.045,E2 32389.045} C_VEL
LIN {X 0,Y 681.113,Z 762.785,A -85,B 0,C 180,E1 32385.765,E2 32385.765} C_VEL
LIN {X 0,Y 683.969,Z 719.936,A -85,B 0,C 180,E1 32382.517,E2 32382.517} C_VEL
LIN {X 0,Y 685.933,Z 686.583,A -85,B 0,C 180,E1 32379.839,E2 32379.839} C_VEL
LIN {X 0,Y 686.088,Z 680.55,A -85,B 0,C 180,E1 32379.326,E2 32379.326} C_VEL
LIN {X 0,Y 680.857,Z 667.611,A -85,B 0,C 180,E1 32377.644,E2 32377.644} C_VEL
LIN {X 0,Y 676.485,Z 657.439,A -85,B 0,C 180,E1 32376.19,E2 32376.19} C_VEL
LIN {X 0,Y 674.866,Z 654.159,A -85,B 0,C 180,E1 32375.666,E2 32375.666} C_VEL
LIN {X 0,Y 672.725,Z 649.764,A -85,B 0,C 180,E1 32374.938,E2 32374.938} C_VEL
LIN {X 0,Y 672.573,Z 648.891,A -85,B 0,C 180,E1 32374.79,E2 32374.79} C_VEL
LIN {X 0,Y 672.568,Z 648.891,A -85,B 0,C 180,E1 32371.786,E2 32371.786} C_VEL
LIN {X 0,Y 672.567,Z 648.891,A -85,B 0,C 180,E1 32368.844,E2 32368.844} C_VEL
LIN {X 0,Y 672.573,Z 648.893,A -85,B 0,C 180,E1 32365.898,E2 32365.898} C_VEL
LIN {X 0,Y 672.577,Z 648.889,A -85,B 0,C 180,E1 32362.827,E2 32362.827} C_VEL
LIN {X 0,Y 672.58,Z 648.891,A -85,B 0,C 180,E1 32359.819,E2 32359.819} C_VEL
LIN {X 0,Y 672.583,Z 648.889,A -85,B 0,C 180,E1 32356.737,E2 32356.737} C_VEL
LIN {X 0,Y 672.602,Z 649.1,A -85,B 0,C 180,E1 32356.472,E2 32356.472} C_VEL
LIN {X 0,Y 674.035,Z 652.591,A -85,B 0,C 180,E1 32356.032,E2 32356.032} C_VEL
LIN {X 0,Y 675.099,Z 654.645,A -85,B 0,C 180,E1 32355.765,E2 32355.765} C_VEL
LIN {X 0,Y 679.036,Z 662.893,A -85,B 0,C 180,E1 32354.785,E2 32354.785} C_VEL
LIN {X 0,Y 684.203,Z 674.888,A -85,B 0,C 180,E1 32353.543,E2 32353.543} C_VEL
LIN {X 0,Y 684.571,Z 676.51,A -85,B 0,C 180,E1 32353.408,E2 32353.408} C_VEL
LIN {X 0,Y 681.741,Z 721.829,A -85,B 0,C 180,E1 32350.817,E2 32350.817} C_VEL
LIN {X 0,Y 680.226,Z 768.092,A -85,B 0,C 180,E1 32348.284,E2 32348.284} C_VEL
LIN {X 0,Y 681.733,Z 787.898,A -85,B 0,C 180,E1 32347.141,E2 32347.141} C_VEL
LIN {X 0,Y 684.704,Z 802.133,A -85,B 0,C 180,E1 32346.257,E2 32346.257} C_VEL
LIN {X 0,Y 688.914,Z 813.586,A -85,B 0,C 180,E1 32345.488,E2 32345.488} C_VEL
LIN {X 0,Y 694.138,Z 823.022,A -85,B 0,C 180,E1 32344.807,E2 32344.807} C_VEL
LIN {X 0,Y 700.748,Z 831.379,A -85,B 0,C 180,E1 32344.147,E2 32344.147} C_VEL
LIN {X 0,Y 708.766,Z 838.636,A -85,B 0,C 180,E1 32343.513,E2 32343.513} C_VEL
LIN {X 0,Y 718.181,Z 844.633,A -85,B 0,C 180,E1 32342.909,E2 32342.909} C_VEL
LIN {X 0,Y 725.483,Z 847.867,A -85,B 0,C 180,E1 32342.49,E2 32342.49} C_VEL
LIN {X 0,Y 729.828,Z 848.846,A -85,B 0,C 180,E1 32342.147,E2 32342.147} C_VEL
LIN {X 0,Y 733.548,Z 848.747,A -85,B 0,C 180,E1 32341.726,E2 32341.726} C_VEL
LIN {X 0,Y 736.159,Z 847.477,A -85,B 0,C 180,E1 32341.253,E2 32341.253} C_VEL
LIN {X 0,Y 737.301,Z 845.137,A -85,B 0,C 180,E1 32340.769,E2 32340.769} C_VEL
LIN {X 0,Y 736.808,Z 841.839,A -85,B 0,C 180,E1 32340.295,E2 32340.295} C_VEL
LIN {X 0,Y 734.755,Z 837.976,A -85,B 0,C 180,E1 32339.893,E2 32339.893} C_VEL
LIN {X 0,Y 729.701,Z 829.002,A -85,B 0,C 180,E1 32339.195,E2 32339.195} C_VEL
LIN {X 0,Y 729.229,Z 828.212,A -85,B 0,C 180,E1 32339.129,E2 32339.129} C_VEL
LIN {X 0,Y 725.954,Z 862.685,A -85,B 0,C 180,E1 32338.662,E2 32338.662} C_VEL
LIN {X 0,Y 723.836,Z 878.148,A -85,B 0,C 180,E1 32338.353,E2 32338.353} C_VEL
LIN {X 0,Y 723.137,Z 882.667,A -85,B 0,C 180,E1 32338.251,E2 32338.251} C_VEL
LIN {X 0,Y 721,Z 901.669,A -85,B 0,C 180,E1 32338.113,E2 32338.113} C_VEL
LIN {X 0,Y 716.862,Z 920.777,A -85,B 0,C 180,E1 32337.997,E2 32337.997} C_VEL
LIN {X 0,Y 710.772,Z 939.601,A -85,B 0,C 180,E1 32337.861,E2 32337.861} C_VEL
LIN {X 0,Y 703.622,Z 956.902,A -85,B 0,C 180,E1 32337.652,E2 32337.652} C_VEL
LIN {X 0,Y 696.934,Z 972.275,A -85,B 0,C 180,E1 32337.328,E2 32337.328} C_VEL
LIN {X 0,Y 692.505,Z 984.172,A -85,B 0,C 180,E1 32336.959,E2 32336.959} C_VEL
LIN {X 0,Y 690.889,Z 988.857,A -85,B 0,C 180,E1 32336.799,E2 32336.799} C_VEL
LIN {X 0,Y 685.945,Z 1000.609,A -85,B 0,C 180,E1 32336.439,E2 32336.439} C_VEL
LIN {X 0,Y 680.342,Z 1019.756,A -85,B 0,C 180,E1 32335.692,E2 32335.692} C_VEL
LIN {X 0,Y 679.442,Z 1024.444,A -85,B 0,C 180,E1 32335.514,E2 32335.514} C_VEL
LIN {X 0,Y 679.093,Z 1065.122,A -85,B 0,C 180,E1 32335.028,E2 32335.028} C_VEL
LIN {X 0,Y 678.649,Z 1087.889,A -85,B 0,C 180,E1 32334.595,E2 32334.595} C_VEL
LIN {X 0,Y 678.098,Z 1109.851,A -85,B 0,C 180,E1 32334.013,E2 32334.013} C_VEL
LIN {X 0,Y 677.477,Z 1130.775,A -85,B 0,C 180,E1 32333.298,E2 32333.298} C_VEL
LIN {X 0,Y 676.732,Z 1151.71,A -85,B 0,C 180,E1 32332.407,E2 32332.407} C_VEL
LIN {X 0,Y 675.983,Z 1171.745,A -85,B 0,C 180,E1 32331.373,E2 32331.373} C_VEL
LIN {X 0,Y 675.211,Z 1191.18,A -85,B 0,C 180,E1 32330.183,E2 32330.183} C_VEL
LIN {X 0,Y 674.563,Z 1207.163,A -85,B 0,C 180,E1 32329.031,E2 32329.031} C_VEL
LIN {X 0,Y 673.98,Z 1222.202,A -85,B 0,C 180,E1 32327.794,E2 32327.794} C_VEL
LIN {X 0,Y 673.375,Z 1238.736,A -85,B 0,C 180,E1 32326.209,E2 32326.209} C_VEL
LIN {X 0,Y 672.926,Z 1252.017,A -85,B 0,C 180,E1 32324.718,E2 32324.718} C_VEL
LIN {X 0,Y 672.566,Z 1264.752,A -85,B 0,C 180,E1 32323.059,E2 32323.059} C_VEL
LIN {X 0,Y 672.293,Z 1275.329,A -85,B 0,C 180,E1 32321.407,E2 32321.407} C_VEL
LIN {X 0,Y 672.128,Z 1284.241,A -85,B 0,C 180,E1 32319.763,E2 32319.763} C_VEL
LIN {X 0,Y 671.998,Z 1292.587,A -85,B 0,C 180,E1 32317.867,E2 32317.867} C_VEL
LIN {X 0,Y 671.94,Z 1298.384,A -85,B 0,C 180,E1 32316.149,E2 32316.149} C_VEL
LIN {X 0,Y 671.921,Z 1302.586,A -85,B 0,C 180,E1 32314.522,E2 32314.522} C_VEL
LIN {X 0,Y 671.91,Z 1305.936,A -85,B 0,C 180,E1 32312.558,E2 32312.558} C_VEL
LIN {X 0,Y 671.905,Z 1307.316,A -85,B 0,C 180,E1 32310.681,E2 32310.681} C_VEL
LIN {X 0,Y 671.916,Z 1307.204,A -85,B 0,C 180,E1 32308.976,E2 32308.976} C_VEL
LIN {X 0,Y 671.918,Z 1305.232,A -85,B 0,C 180,E1 32306.928,E2 32306.928} C_VEL
LIN {X 0,Y 671.917,Z 1301.801,A -85,B 0,C 180,E1 32305.133,E2 32305.133} C_VEL
LIN {X 0,Y 671.951,Z 1296.588,A -85,B 0,C 180,E1 32303.248,E2 32303.248} C_VEL
LIN {X 0,Y 672.034,Z 1289.75,A -85,B 0,C 180,E1 32301.442,E2 32301.442} C_VEL
LIN {X 0,Y 672.162,Z 1281.601,A -85,B 0,C 180,E1 32299.716,E2 32299.716} C_VEL
LIN {X 0,Y 672.397,Z 1271.085,A -85,B 0,C 180,E1 32297.896,E2 32297.896} C_VEL
LIN {X 0,Y 672.67,Z 1260.23,A -85,B 0,C 180,E1 32296.328,E2 32296.328} C_VEL
LIN {X 0,Y 673.078,Z 1247.59,A -85,B 0,C 180,E1 32294.754,E2 32294.754} C_VEL
LIN {X 0,Y 673.596,Z 1232.59,A -85,B 0,C 180,E1 32293.174,E2 32293.174} C_VEL
LIN {X 0,Y 674.106,Z 1218.581,A -85,B 0,C 180,E1 32291.895,E2 32291.895} C_VEL
LIN {X 0,Y 674.776,Z 1202.194,A -85,B 0,C 180,E1 32290.588,E2 32290.588} C_VEL
LIN {X 0,Y 675.495,Z 1184.305,A -85,B 0,C 180,E1 32289.371,E2 32289.371} C_VEL
LIN {X 0,Y 676.231,Z 1165.036,A -85,B 0,C 180,E1 32288.259,E2 32288.259} C_VEL
LIN {X 0,Y 676.979,Z 1144.746,A -85,B 0,C 180,E1 32287.279,E2 32287.279} C_VEL
LIN {X 0,Y 677.702,Z 1123.373,A -85,B 0,C 180,E1 32286.431,E2 32286.431} C_VEL
LIN {X 0,Y 678.333,Z 1101.62,A -85,B 0,C 180,E1 32285.747,E2 32285.747} C_VEL
LIN {X 0,Y 678.842,Z 1079.304,A -85,B 0,C 180,E1 32285.222,E2 32285.222} C_VEL
LIN {X 0,Y 679.196,Z 1056.92,A -85,B 0,C 180,E1 32284.857,E2 32284.857} C_VEL
LIN {X 0,Y 679.532,Z 1023.332,A -85,B 0,C 180,E1 32284.46,E2 32284.46} C_VEL
LIN {X 0,Y 682.332,Z 1012.423,A -85,B 0,C 180,E1 32284.013,E2 32284.013} C_VEL
LIN {X 0,Y 686.675,Z 998.631,A -85,B 0,C 180,E1 32283.492,E2 32283.492} C_VEL
LIN {X 0,Y 691.708,Z 986.909,A -85,B 0,C 180,E1 32283.144,E2 32283.144} C_VEL
LIN {X 0,Y 695.291,Z 976.337,A -85,B 0,C 180,E1 32282.785,E2 32282.785} C_VEL
LIN {X 0,Y 701.615,Z 961.461,A -85,B 0,C 180,E1 32282.428,E2 32282.428} C_VEL
LIN {X 0,Y 709.137,Z 943.817,A -85,B 0,C 180,E1 32282.178,E2 32282.178} C_VEL
LIN {X 0,Y 715.709,Z 924.871,A -85,B 0,C 180,E1 32282.029,E2 32282.029} C_VEL
LIN {X 0,Y 720.266,Z 905.856,A -85,B 0,C 180,E1 32281.913,E2 32281.913} C_VEL
LIN {X 0,Y 722.83,Z 886.825,A -85,B 0,C 180,E1 32281.783,E2 32281.783} C_VEL
LIN {X 0,Y 723.404,Z 880.429,A -85,B 0,C 180,E1 32281.71,E2 32281.71} C_VEL
LIN {X 0,Y 725.382,Z 867.525,A -85,B 0,C 180,E1 32281.421,E2 32281.421} C_VEL
LIN {X 0,Y 728.347,Z 838.415,A -85,B 0,C 180,E1 32280.996,E2 32280.996} C_VEL
LIN {X 0,Y 729.288,Z 828.143,A -85,B 0,C 180,E1 32280.863,E2 32280.863} C_VEL
LIN {X 0,Y 734.271,Z 837.227,A -85,B 0,C 180,E1 32280.173,E2 32280.173} C_VEL
LIN {X 0,Y 736.625,Z 841.364,A -85,B 0,C 180,E1 32279.761,E2 32279.761} C_VEL
LIN {X 0,Y 737.339,Z 844.609,A -85,B 0,C 180,E1 32279.317,E2 32279.317} C_VEL
LIN {X 0,Y 736.539,Z 847.058,A -85,B 0,C 180,E1 32278.853,E2 32278.853} C_VEL
LIN {X 0,Y 734.27,Z 848.553,A -85,B 0,C 180,E1 32278.38,E2 32278.38} C_VEL
LIN {X 0,Y 730.494,Z 848.91,A -85,B 0,C 180,E1 32277.917,E2 32277.917} C_VEL
LIN {X 0,Y 726.245,Z 848.105,A -85,B 0,C 180,E1 32277.563,E2 32277.563} C_VEL
LIN {X 0,Y 716.133,Z 843.718,A -85,B 0,C 180,E1 32276.903,E2 32276.903} C_VEL
LIN {X 0,Y 707.335,Z 837.795,A -85,B 0,C 180,E1 32276.223,E2 32276.223} C_VEL
LIN {X 0,Y 699.922,Z 830.577,A -85,B 0,C 180,E1 32275.517,E2 32275.517} C_VEL
LIN {X 0,Y 693.63,Z 821.626,A -85,B 0,C 180,E1 32274.749,E2 32274.749} C_VEL
LIN {X 0,Y 688.585,Z 810.637,A -85,B 0,C 180,E1 32273.91,E2 32273.91} C_VEL
LIN {X 0,Y 685.132,Z 797.93,A -85,B 0,C 180,E1 32273.038,E2 32273.038} C_VEL
LIN {X 0,Y 683.17,Z 782.404,A -85,B 0,C 180,E1 32272.068,E2 32272.068} C_VEL
LIN {X 0,Y 682.751,Z 762.376,A -85,B 0,C 180,E1 32270.913,E2 32270.913} C_VEL
LIN {X 0,Y 684.578,Z 711.396,A -85,B 0,C 180,E1 32268.069,E2 32268.069} C_VEL
LIN {X 0,Y 685.792,Z 678.697,A -85,B 0,C 180,E1 32266.196,E2 32266.196} C_VEL
LIN {X 0,Y 675.108,Z 655.225,A -85,B 0,C 180,E1 32263.998,E2 32263.998} C_VEL
LIN {X 0,Y 672.634,Z 649.215,A -85,B 0,C 180,E1 32263.433,E2 32263.433} C_VEL
LIN {X 0,Y 672.589,Z 648.889,A -85,B 0,C 180,E1 32263.367,E2 32263.367} C_VEL
LIN {X 0,Y 672.574,Z 648.891,A -85,B 0,C 180,E1 32260.293,E2 32260.293} C_VEL
LIN {X 0,Y 672.567,Z 648.892,A -85,B 0,C 180,E1 32257.309,E2 32257.309} C_VEL
LIN {X 0,Y 672.586,Z 648.892,A -85,B 0,C 180,E1 32254.251,E2 32254.251} C_VEL
LIN {X 0,Y 672.591,Z 649.048,A -85,B 0,C 180,E1 32253.129,E2 32253.129} C_VEL
LIN {X 0,Y 678.478,Z 668.795,A -85,B 0,C 180,E1 32251.249,E2 32251.249} C_VEL
LIN {X 0,Y 677.877,Z 701.997,A -85,B 0,C 180,E1 32248.596,E2 32248.596} C_VEL
LIN {X 0,Y 681.1,Z 717.029,A -85,B 0,C 180,E1 32248.259,E2 32248.259} C_VEL
LIN {X 0,Y 679.801,Z 907.308,A -85,B 0,C 180,E1 32246.105,E2 32246.105} C_VEL
LIN {X 0,Y 679.134,Z 1002.306,A -85,B 0,C 180,E1 32245.022,E2 32245.022} C_VEL
LIN {X 0,Y 678.693,Z 1025.143,A -85,B 0,C 180,E1 32244.61,E2 32244.61} C_VEL
LIN {X 0,Y 678.218,Z 1046.131,A -85,B 0,C 180,E1 32244.08,E2 32244.08} C_VEL
LIN {X 0,Y 677.564,Z 1067.328,A -85,B 0,C 180,E1 32243.379,E2 32243.379} C_VEL
LIN {X 0,Y 676.87,Z 1087.731,A -85,B 0,C 180,E1 32242.541,E2 32242.541} C_VEL
LIN {X 0,Y 676.136,Z 1107.529,A -85,B 0,C 180,E1 32241.561,E2 32241.561} C_VEL
LIN {X 0,Y 675.408,Z 1126.436,A -85,B 0,C 180,E1 32240.45,E2 32240.45} C_VEL
LIN {X 0,Y 674.686,Z 1144.265,A -85,B 0,C 180,E1 32239.209,E2 32239.209} C_VEL
LIN {X 0,Y 674.016,Z 1161.171,A -85,B 0,C 180,E1 32237.839,E2 32237.839} C_VEL
LIN {X 0,Y 673.447,Z 1176.608,A -85,B 0,C 180,E1 32236.386,E2 32236.386} C_VEL
LIN {X 0,Y 672.972,Z 1190.981,A -85,B 0,C 180,E1 32234.807,E2 32234.807} C_VEL
LIN {X 0,Y 672.586,Z 1203.753,A -85,B 0,C 180,E1 32233.147,E2 32233.147} C_VEL
LIN {X 0,Y 672.305,Z 1215.063,A -85,B 0,C 180,E1 32231.409,E2 32231.409} C_VEL
LIN {X 0,Y 672.118,Z 1224.459,A -85,B 0,C 180,E1 32229.678,E2 32229.678} C_VEL
LIN {X 0,Y 672.007,Z 1232.395,A -85,B 0,C 180,E1 32227.868,E2 32227.868} C_VEL
LIN {X 0,Y 671.949,Z 1238.52,A -85,B 0,C 180,E1 32226.065,E2 32226.065} C_VEL
LIN {X 0,Y 671.916,Z 1243.06,A -85,B 0,C 180,E1 32224.267,E2 32224.267} C_VEL
LIN {X 0,Y 671.906,Z 1245.949,A -85,B 0,C 180,E1 32222.473,E2 32222.473} C_VEL
LIN {X 0,Y 671.912,Z 1247.339,A -85,B 0,C 180,E1 32220.597,E2 32220.597} C_VEL
LIN {X 0,Y 671.903,Z 1247.184,A -85,B 0,C 180,E1 32218.806,E2 32218.806} C_VEL
LIN {X 0,Y 671.901,Z 1245.281,A -85,B 0,C 180,E1 32216.929,E2 32216.929} C_VEL
LIN {X 0,Y 671.921,Z 1241.714,A -85,B 0,C 180,E1 32215.049,E2 32215.049} C_VEL
LIN {X 0,Y 671.967,Z 1236.733,A -85,B 0,C 180,E1 32213.249,E2 32213.249} C_VEL
LIN {X 0,Y 672.026,Z 1229.949,A -85,B 0,C 180,E1 32211.443,E2 32211.443} C_VEL
LIN {X 0,Y 672.167,Z 1221.373,A -85,B 0,C 180,E1 32209.63,E2 32209.63} C_VEL
LIN {X 0,Y 672.382,Z 1211.392,A -85,B 0,C 180,E1 32207.896,E2 32207.896} C_VEL
LIN {X 0,Y 672.689,Z 1199.971,A -85,B 0,C 180,E1 32206.242,E2 32206.242} C_VEL
LIN {X 0,Y 673.104,Z 1186.572,A -85,B 0,C 180,E1 32204.598,E2 32204.598} C_VEL
LIN {X 0,Y 673.644,Z 1171.258,A -85,B 0,C 180,E1 32202.998,E2 32202.998} C_VEL
LIN {X 0,Y 674.254,Z 1155.528,A -85,B 0,C 180,E1 32201.587,E2 32201.587} C_VEL
LIN {X 0,Y 674.927,Z 1138.241,A -85,B 0,C 180,E1 32200.258,E2 32200.258} C_VEL
LIN {X 0,Y 675.621,Z 1120.625,A -85,B 0,C 180,E1 32199.104,E2 32199.104} C_VEL
LIN {X 0,Y 676.402,Z 1100.691,A -85,B 0,C 180,E1 32197.992,E2 32197.992} C_VEL
LIN {X 0,Y 677.086,Z 1081.746,A -85,B 0,C 180,E1 32197.1,E2 32197.1} C_VEL
LIN {X 0,Y 677.778,Z 1061.023,A -85,B 0,C 180,E1 32196.307,E2 32196.307} C_VEL
LIN {X 0,Y 678.364,Z 1039.234,A -85,B 0,C 180,E1 32195.642,E2 32195.642} C_VEL
LIN {X 0,Y 678.877,Z 1017.268,A -85,B 0,C 180,E1 32195.138,E2 32195.138} C_VEL
LIN {X 0,Y 678.959,Z 1011.799,A -85,B 0,C 180,E1 32195.038,E2 32195.038} C_VEL
LIN {X 0,Y 678.212,Z 1004.299,A -85,B 0,C 180,E1 32194.878,E2 32194.878} C_VEL
LIN {X 0,Y 672.697,Z 984.536,A -85,B 0,C 180,E1 32194.413,E2 32194.413} C_VEL
LIN {X 0,Y 672.045,Z 978.015,A -85,B 0,C 180,E1 32194.316,E2 32194.316} C_VEL
LIN {X 0,Y 673.936,Z 728.777,A -85,B 0,C 180,E1 32191.47,E2 32191.47} C_VEL
LIN {X 0,Y 673.847,Z 716.597,A -85,B 0,C 180,E1 32191.311,E2 32191.311} C_VEL
LIN {X 0,Y 670.236,Z 700.558,A -85,B 0,C 180,E1 32190.921,E2 32190.921} C_VEL
LIN {X 0,Y 671.096,Z 670.986,A -85,B 0,C 180,E1 32188.457,E2 32188.457} C_VEL
LIN {X 0,Y 664.643,Z 649.882,A -85,B 0,C 180,E1 32186.281,E2 32186.281} C_VEL
LIN {X 0,Y 664.645,Z 649.876,A -85,B 0,C 180,E1 32183.112,E2 32183.112} C_VEL
LIN {X 0,Y 664.649,Z 649.877,A -85,B 0,C 180,E1 32179.918,E2 32179.918} C_VEL
LIN {X 0,Y 664.644,Z 649.879,A -85,B 0,C 180,E1 32176.803,E2 32176.803} C_VEL
LIN {X 0,Y 664.65,Z 649.876,A -85,B 0,C 180,E1 32173.646,E2 32173.646} C_VEL
LIN {X 0,Y 664.649,Z 649.874,A -85,B 0,C 180,E1 32170.534,E2 32170.534} C_VEL
LIN {X 0,Y 664.641,Z 649.873,A -85,B 0,C 180,E1 32167.321,E2 32167.321} C_VEL
LIN {X 0,Y 664.645,Z 649.878,A -85,B 0,C 180,E1 32164.24,E2 32164.24} C_VEL
LIN {X 0,Y 664.652,Z 649.875,A -85,B 0,C 180,E1 32161.13,E2 32161.13} C_VEL
LIN {X 0,Y 664.643,Z 649.872,A -85,B 0,C 180,E1 32157.983,E2 32157.983} C_VEL
LIN {X 0,Y 664.639,Z 649.875,A -85,B 0,C 180,E1 32154.818,E2 32154.818} C_VEL
LIN {X 0,Y 664.642,Z 649.88,A -85,B 0,C 180,E1 32151.722,E2 32151.722} C_VEL
LIN {X 0,Y 664.651,Z 649.875,A -85,B 0,C 180,E1 32148.599,E2 32148.599} C_VEL
LIN {X 0,Y 664.639,Z 649.874,A -85,B 0,C 180,E1 32145.444,E2 32145.444} C_VEL
LIN {X 0,Y 664.64,Z 649.873,A -85,B 0,C 180,E1 32142.336,E2 32142.336} C_VEL
LIN {X 0,Y 664.641,Z 649.876,A -85,B 0,C 180,E1 32139.264,E2 32139.264} C_VEL
LIN {X 0,Y 664.651,Z 649.875,A -85,B 0,C 180,E1 32136.219,E2 32136.219} C_VEL
LIN {X 0,Y 664.641,Z 649.872,A -85,B 0,C 180,E1 32133.019,E2 32133.019} C_VEL
LIN {X 0,Y 664.645,Z 649.871,A -85,B 0,C 180,E1 32129.915,E2 32129.915} C_VEL
LIN {X 0,Y 664.642,Z 649.878,A -85,B 0,C 180,E1 32126.81,E2 32126.81} C_VEL
LIN {X 0,Y 664.652,Z 649.876,A -85,B 0,C 180,E1 32123.696,E2 32123.696} C_VEL
LIN {X 0,Y 664.642,Z 649.873,A -85,B 0,C 180,E1 32120.563,E2 32120.563} C_VEL
LIN {X 0,Y 664.641,Z 649.875,A -85,B 0,C 180,E1 32117.402,E2 32117.402} C_VEL
LIN {X 0,Y 664.643,Z 649.88,A -85,B 0,C 180,E1 32114.29,E2 32114.29} C_VEL
LIN {X 0,Y 664.651,Z 649.876,A -85,B 0,C 180,E1 32111.221,E2 32111.221} C_VEL
LIN {X 0,Y 664.642,Z 649.874,A -85,B 0,C 180,E1 32108.002,E2 32108.002} C_VEL
LIN {X 0,Y 664.642,Z 649.873,A -85,B 0,C 180,E1 32104.899,E2 32104.899} C_VEL
LIN {X 0,Y 664.646,Z 649.88,A -85,B 0,C 180,E1 32101.813,E2 32101.813} C_VEL
LIN {X 0,Y 664.653,Z 649.878,A -85,B 0,C 180,E1 32098.704,E2 32098.704} C_VEL
LIN {X 0,Y 664.641,Z 649.877,A -85,B 0,C 180,E1 32095.53,E2 32095.53} C_VEL
LIN {X 0,Y 664.645,Z 649.877,A -85,B 0,C 180,E1 32092.45,E2 32092.45} C_VEL
LIN {X 0,Y 664.644,Z 649.879,A -85,B 0,C 180,E1 32089.308,E2 32089.308} C_VEL
LIN {X 0,Y 664.651,Z 649.878,A -85,B 0,C 180,E1 32086.213,E2 32086.213} C_VEL
LIN {X 0,Y 664.639,Z 649.879,A -85,B 0,C 180,E1 32083.02,E2 32083.02} C_VEL
LIN {X 0,Y 664.654,Z 649.926,A -85,B 0,C 180,E1 32082.312,E2 32082.312} C_VEL
LIN {X 0,Y 672.925,Z 674.135,A -85,B 0,C 180,E1 32080.009,E2 32080.009} C_VEL
LIN {X 0,Y 671.704,Z 714.756,A -85,B 0,C 180,E1 32077.075,E2 32077.075} C_VEL
LIN {X 0,Y 670.221,Z 760.12,A -85,B 0,C 180,E1 32073.864,E2 32073.864} C_VEL
LIN {X 0,Y 668.865,Z 805.549,A -85,B 0,C 180,E1 32070.698,E2 32070.698} C_VEL
LIN {X 0,Y 667.624,Z 852.441,A -85,B 0,C 180,E1 32067.47,E2 32067.47} C_VEL
LIN {X 0,Y 666.724,Z 895.174,A -85,B 0,C 180,E1 32064.585,E2 32064.585} C_VEL
LIN {X 0,Y 667.276,Z 902.203,A -85,B 0,C 180,E1 32064.48,E2 32064.48} C_VEL
LIN {X 0,Y 666.784,Z 963.539,A -85,B 0,C 180,E1 32063.761,E2 32063.761} C_VEL
LIN {X 0,Y 666.321,Z 1032.216,A -85,B 0,C 180,E1 32062.944,E2 32062.944} C_VEL
LIN {X 0,Y 666.189,Z 1047.988,A -85,B 0,C 180,E1 32062.657,E2 32062.657} C_VEL
LIN {X 0,Y 666.005,Z 1063.225,A -85,B 0,C 180,E1 32062.231,E2 32062.231} C_VEL
LIN {X 0,Y 665.716,Z 1079.488,A -85,B 0,C 180,E1 32061.591,E2 32061.591} C_VEL
LIN {X 0,Y 665.398,Z 1093.468,A -85,B 0,C 180,E1 32060.863,E2 32060.863} C_VEL
LIN {X 0,Y 665.13,Z 1106.18,A -85,B 0,C 180,E1 32060.028,E2 32060.028} C_VEL
LIN {X 0,Y 664.873,Z 1117.207,A -85,B 0,C 180,E1 32059.138,E2 32059.138} C_VEL
LIN {X 0,Y 664.636,Z 1127.323,A -85,B 0,C 180,E1 32058.145,E2 32058.145} C_VEL
LIN {X 0,Y 664.399,Z 1137.552,A -85,B 0,C 180,E1 32056.885,E2 32056.885} C_VEL
LIN {X 0,Y 664.257,Z 1145.42,A -85,B 0,C 180,E1 32055.631,E2 32055.631} C_VEL
LIN {X 0,Y 664.171,Z 1151.041,A -85,B 0,C 180,E1 32054.472,E2 32054.472} C_VEL
LIN {X 0,Y 664.123,Z 1155.507,A -85,B 0,C 180,E1 32053.229,E2 32053.229} C_VEL
LIN {X 0,Y 664.097,Z 1158.731,A -85,B 0,C 180,E1 32051.867,E2 32051.867} C_VEL
LIN {X 0,Y 664.089,Z 1160.352,A -85,B 0,C 180,E1 32050.322,E2 32050.322} C_VEL
LIN {X 0,Y 664.103,Z 1159.973,A -85,B 0,C 180,E1 32048.921,E2 32048.921} C_VEL
LIN {X 0,Y 664.124,Z 1158.08,A -85,B 0,C 180,E1 32047.614,E2 32047.614} C_VEL
LIN {X 0,Y 664.167,Z 1154.67,A -85,B 0,C 180,E1 32046.31,E2 32046.31} C_VEL
LIN {X 0,Y 664.258,Z 1149.218,A -85,B 0,C 180,E1 32044.922,E2 32044.922} C_VEL
LIN {X 0,Y 664.418,Z 1141.601,A -85,B 0,C 180,E1 32043.537,E2 32043.537} C_VEL
LIN {X 0,Y 664.61,Z 1133.633,A -85,B 0,C 180,E1 32042.414,E2 32042.414} C_VEL
LIN {X 0,Y 664.875,Z 1123.724,A -85,B 0,C 180,E1 32041.293,E2 32041.293} C_VEL
LIN {X 0,Y 665.213,Z 1110.715,A -85,B 0,C 180,E1 32040.129,E2 32040.129} C_VEL
LIN {X 0,Y 665.514,Z 1097.814,A -85,B 0,C 180,E1 32039.225,E2 32039.225} C_VEL
LIN {X 0,Y 665.804,Z 1084.845,A -85,B 0,C 180,E1 32038.494,E2 32038.494} C_VEL
LIN {X 0,Y 666.113,Z 1070.211,A -85,B 0,C 180,E1 32037.849,E2 32037.849} C_VEL
LIN {X 0,Y 666.345,Z 1053.362,A -85,B 0,C 180,E1 32037.312,E2 32037.312} C_VEL
LIN {X 0,Y 666.483,Z 1037.329,A -85,B 0,C 180,E1 32036.977,E2 32036.977} C_VEL
LIN {X 0,Y 667.952,Z 898.863,A -85,B 0,C 180,E1 32035.178,E2 32035.178} C_VEL
LIN {X 0,Y 669.485,Z 855.838,A -85,B 0,C 180,E1 32032.145,E2 32032.145} C_VEL
LIN {X 0,Y 671.674,Z 808.432,A -85,B 0,C 180,E1 32028.711,E2 32028.711} C_VEL
LIN {X 0,Y 674.34,Z 763.4,A -85,B 0,C 180,E1 32025.356,E2 32025.356} C_VEL
LIN {X 0,Y 677.513,Z 720.211,A -85,B 0,C 180,E1 32022.034,E2 32022.034} C_VEL
LIN {X 0,Y 679.775,Z 685.017,A -85,B 0,C 180,E1 32019.148,E2 32019.148} C_VEL
LIN {X 0,Y 674.071,Z 670.525,A -85,B 0,C 180,E1 32017.222,E2 32017.222} C_VEL
LIN {X 0,Y 670.179,Z 662.032,A -85,B 0,C 180,E1 32015.931,E2 32015.931} C_VEL
LIN {X 0,Y 668.242,Z 657.931,A -85,B 0,C 180,E1 32015.26,E2 32015.26} C_VEL
LIN {X 0,Y 666.402,Z 653.971,A -85,B 0,C 180,E1 32014.585,E2 32014.585} C_VEL
LIN {X 0,Y 664.725,Z 650.469,A -85,B 0,C 180,E1 32013.945,E2 32013.945} C_VEL
LIN {X 0,Y 664.632,Z 649.879,A -85,B 0,C 180,E1 32013.845,E2 32013.845} C_VEL
LIN {X 0,Y 664.629,Z 649.88,A -85,B 0,C 180,E1 32010.828,E2 32010.828} C_VEL
LIN {X 0,Y 664.629,Z 649.879,A -85,B 0,C 180,E1 32007.821,E2 32007.821} C_VEL
LIN {X 0,Y 664.631,Z 649.88,A -85,B 0,C 180,E1 32004.773,E2 32004.773} C_VEL
LIN {X 0,Y 664.633,Z 649.882,A -85,B 0,C 180,E1 32001.746,E2 32001.746} C_VEL
LIN {X 0,Y 664.639,Z 649.878,A -85,B 0,C 180,E1 31998.667,E2 31998.667} C_VEL
LIN {X 0,Y 664.662,Z 650.125,A -85,B 0,C 180,E1 31997.308,E2 31997.308} C_VEL
LIN {X 0,Y 666.165,Z 653.667,A -85,B 0,C 180,E1 31996.808,E2 31996.808} C_VEL
LIN {X 0,Y 667.207,Z 655.445,A -85,B 0,C 180,E1 31996.538,E2 31996.538} C_VEL
LIN {X 0,Y 671.262,Z 663.738,A -85,B 0,C 180,E1 31995.445,E2 31995.445} C_VEL
LIN {X 0,Y 676.566,Z 675.874,A -85,B 0,C 180,E1 31994.089,E2 31994.089} C_VEL
LIN {X 0,Y 678.064,Z 679.88,A -85,B 0,C 180,E1 31993.696,E2 31993.696} C_VEL
LIN {X 0,Y 674.868,Z 725.289,A -85,B 0,C 180,E1 31991.049,E2 31991.049} C_VEL
LIN {X 0,Y 673.142,Z 770.204,A -85,B 0,C 180,E1 31988.543,E2 31988.543} C_VEL
LIN {X 0,Y 674.49,Z 789.893,A -85,B 0,C 180,E1 31987.383,E2 31987.383} C_VEL
LIN {X 0,Y 677.438,Z 804.754,A -85,B 0,C 180,E1 31986.446,E2 31986.446} C_VEL
LIN {X 0,Y 681.623,Z 816.606,A -85,B 0,C 180,E1 31985.641,E2 31985.641} C_VEL
LIN {X 0,Y 687.308,Z 827.191,A -85,B 0,C 180,E1 31984.864,E2 31984.864} C_VEL
LIN {X 0,Y 694.551,Z 836.441,A -85,B 0,C 180,E1 31984.128,E2 31984.128} C_VEL
LIN {X 0,Y 703.284,Z 844.37,A -85,B 0,C 180,E1 31983.429,E2 31983.429} C_VEL
LIN {X 0,Y 713.498,Z 850.886,A -85,B 0,C 180,E1 31982.771,E2 31982.771} C_VEL
LIN {X 0,Y 722.553,Z 854.887,A -85,B 0,C 180,E1 31982.272,E2 31982.272} C_VEL
LIN {X 0,Y 727.046,Z 855.926,A -85,B 0,C 180,E1 31981.946,E2 31981.946} C_VEL
LIN {X 0,Y 730.928,Z 855.932,A -85,B 0,C 180,E1 31981.543,E2 31981.543} C_VEL
LIN {X 0,Y 733.725,Z 854.86,A -85,B 0,C 180,E1 31981.095,E2 31981.095} C_VEL
LIN {X 0,Y 735.215,Z 852.724,A -85,B 0,C 180,E1 31980.612,E2 31980.612} C_VEL
LIN {X 0,Y 735.135,Z 849.72,A -85,B 0,C 180,E1 31980.146,E2 31980.146} C_VEL
LIN {X 0,Y 733.48,Z 846.065,A -85,B 0,C 180,E1 31979.725,E2 31979.725} C_VEL
LIN {X 0,Y 731.845,Z 843.67,A -85,B 0,C 180,E1 31979.494,E2 31979.494} C_VEL
LIN {X 0,Y 728.999,Z 867.736,A -85,B 0,C 180,E1 31979.159,E2 31979.159} C_VEL
LIN {X 0,Y 726.209,Z 882.016,A -85,B 0,C 180,E1 31978.881,E2 31978.881} C_VEL
LIN {X 0,Y 725.437,Z 885.961,A -85,B 0,C 180,E1 31978.829,E2 31978.829} C_VEL
LIN {X 0,Y 721.017,Z 904.659,A -85,B 0,C 180,E1 31978.732,E2 31978.732} C_VEL
LIN {X 0,Y 714.713,Z 922.895,A -85,B 0,C 180,E1 31978.612,E2 31978.612} C_VEL
LIN {X 0,Y 706.677,Z 940.703,A -85,B 0,C 180,E1 31978.427,E2 31978.427} C_VEL
LIN {X 0,Y 697.821,Z 957.621,A -85,B 0,C 180,E1 31978.124,E2 31978.124} C_VEL
LIN {X 0,Y 690.253,Z 972.593,A -85,B 0,C 180,E1 31977.708,E2 31977.708} C_VEL
LIN {X 0,Y 685.674,Z 983.956,A -85,B 0,C 180,E1 31977.305,E2 31977.305} C_VEL
LIN {X 0,Y 684.346,Z 987.574,A -85,B 0,C 180,E1 31977.169,E2 31977.169} C_VEL
LIN {X 0,Y 678.873,Z 999.513,A -85,B 0,C 180,E1 31976.739,E2 31976.739} C_VEL
LIN {X 0,Y 672.945,Z 1019.085,A -85,B 0,C 180,E1 31975.948,E2 31975.948} C_VEL
LIN {X 0,Y 671.955,Z 1024.132,A -85,B 0,C 180,E1 31975.757,E2 31975.757} C_VEL
LIN {X 0,Y 671.674,Z 1065.253,A -85,B 0,C 180,E1 31975.282,E2 31975.282} C_VEL
LIN {X 0,Y 671.269,Z 1088.749,A -85,B 0,C 180,E1 31974.847,E2 31974.847} C_VEL
LIN {X 0,Y 670.775,Z 1109.049,A -85,B 0,C 180,E1 31974.316,E2 31974.316} C_VEL
LIN {X 0,Y 670.088,Z 1130.025,A -85,B 0,C 180,E1 31973.599,E2 31973.599} C_VEL
LIN {X 0,Y 669.301,Z 1150.776,A -85,B 0,C 180,E1 31972.715,E2 31972.715} C_VEL
LIN {X 0,Y 668.468,Z 1170.795,A -85,B 0,C 180,E1 31971.681,E2 31971.681} C_VEL
LIN {X 0,Y 667.604,Z 1190.435,A -85,B 0,C 180,E1 31970.473,E2 31970.473} C_VEL
LIN {X 0,Y 666.894,Z 1206.528,A -85,B 0,C 180,E1 31969.308,E2 31969.308} C_VEL
LIN {X 0,Y 666.25,Z 1221.168,A -85,B 0,C 180,E1 31968.097,E2 31968.097} C_VEL
LIN {X 0,Y 665.617,Z 1237.071,A -85,B 0,C 180,E1 31966.582,E2 31966.582} C_VEL
LIN {X 0,Y 665.1,Z 1250.542,A -85,B 0,C 180,E1 31965.073,E2 31965.073} C_VEL
LIN {X 0,Y 664.707,Z 1262.196,A -85,B 0,C 180,E1 31963.57,E2 31963.57} C_VEL
LIN {X 0,Y 664.376,Z 1274.314,A -85,B 0,C 180,E1 31961.721,E2 31961.721} C_VEL
LIN {X 0,Y 664.161,Z 1283.36,A -85,B 0,C 180,E1 31960.056,E2 31960.056} C_VEL
LIN {X 0,Y 664.036,Z 1291.217,A -85,B 0,C 180,E1 31958.31,E2 31958.31} C_VEL
LIN {X 0,Y 663.954,Z 1297.878,A -85,B 0,C 180,E1 31956.397,E2 31956.397} C_VEL
LIN {X 0,Y 663.918,Z 1302.193,A -85,B 0,C 180,E1 31954.75,E2 31954.75} C_VEL
LIN {X 0,Y 663.917,Z 1305.605,A -85,B 0,C 180,E1 31952.848,E2 31952.848} C_VEL
LIN {X 0,Y 663.917,Z 1307.23,A -85,B 0,C 180,E1 31950.948,E2 31950.948} C_VEL
LIN {X 0,Y 663.906,Z 1307.311,A -85,B 0,C 180,E1 31949.308,E2 31949.308} C_VEL
LIN {X 0,Y 663.912,Z 1305.936,A -85,B 0,C 180,E1 31947.409,E2 31947.409} C_VEL
LIN {X 0,Y 663.922,Z 1302.577,A -85,B 0,C 180,E1 31945.421,E2 31945.421} C_VEL
LIN {X 0,Y 663.947,Z 1298.374,A -85,B 0,C 180,E1 31943.774,E2 31943.774} C_VEL
LIN {X 0,Y 664.024,Z 1292.256,A -85,B 0,C 180,E1 31941.949,E2 31941.949} C_VEL
LIN {X 0,Y 664.155,Z 1283.788,A -85,B 0,C 180,E1 31940.029,E2 31940.029} C_VEL
LIN {X 0,Y 664.359,Z 1274.801,A -85,B 0,C 180,E1 31938.364,E2 31938.364} C_VEL
LIN {X 0,Y 664.695,Z 1262.832,A -85,B 0,C 180,E1 31936.516,E2 31936.516} C_VEL
LIN {X 0,Y 665.075,Z 1251.256,A -85,B 0,C 180,E1 31935.013,E2 31935.013} C_VEL
LIN {X 0,Y 665.546,Z 1238.704,A -85,B 0,C 180,E1 31933.593,E2 31933.593} C_VEL
LIN {X 0,Y 666.214,Z 1222.171,A -85,B 0,C 180,E1 31931.99,E2 31931.99} C_VEL
LIN {X 0,Y 666.843,Z 1207.697,A -85,B 0,C 180,E1 31930.783,E2 31930.783} C_VEL
LIN {X 0,Y 667.577,Z 1191.139,A -85,B 0,C 180,E1 31929.574,E2 31929.574} C_VEL
LIN {X 0,Y 668.436,Z 1171.541,A -85,B 0,C 180,E1 31928.362,E2 31928.362} C_VEL
LIN {X 0,Y 669.258,Z 1151.654,A -85,B 0,C 180,E1 31927.327,E2 31927.327} C_VEL
LIN {X 0,Y 670.027,Z 1131.848,A -85,B 0,C 180,E1 31926.471,E2 31926.471} C_VEL
LIN {X 0,Y 670.733,Z 1110.505,A -85,B 0,C 180,E1 31925.727,E2 31925.727} C_VEL
LIN {X 0,Y 671.263,Z 1089.52,A -85,B 0,C 180,E1 31925.17,E2 31925.17} C_VEL
LIN {X 0,Y 671.686,Z 1066.581,A -85,B 0,C 180,E1 31924.73,E2 31924.73} C_VEL
LIN {X 0,Y 671.984,Z 1032.697,A -85,B 0,C 180,E1 31924.32,E2 31924.32} C_VEL
LIN {X 0,Y 672.119,Z 1023.163,A -85,B 0,C 180,E1 31924.205,E2 31924.205} C_VEL
LIN {X 0,Y 675.201,Z 1011.469,A -85,B 0,C 180,E1 31923.718,E2 31923.718} C_VEL
LIN {X 0,Y 679.876,Z 997.183,A -85,B 0,C 180,E1 31923.159,E2 31923.159} C_VEL
LIN {X 0,Y 685.081,Z 985.864,A -85,B 0,C 180,E1 31922.769,E2 31922.769} C_VEL
LIN {X 0,Y 689.464,Z 974.324,A -85,B 0,C 180,E1 31922.349,E2 31922.349} C_VEL
LIN {X 0,Y 697.037,Z 959.103,A -85,B 0,C 180,E1 31921.911,E2 31921.911} C_VEL
LIN {X 0,Y 705.323,Z 943.372,A -85,B 0,C 180,E1 31921.609,E2 31921.609} C_VEL
LIN {X 0,Y 713.387,Z 926.138,A -85,B 0,C 180,E1 31921.415,E2 31921.415} C_VEL
LIN {X 0,Y 719.702,Z 908.984,A -85,B 0,C 180,E1 31921.293,E2 31921.293} C_VEL
LIN {X 0,Y 724.564,Z 890.44,A -85,B 0,C 180,E1 31921.195,E2 31921.195} C_VEL
LIN {X 0,Y 726.118,Z 882.412,A -85,B 0,C 180,E1 31921.129,E2 31921.129} C_VEL
LIN {X 0,Y 728.874,Z 868.487,A -85,B 0,C 180,E1 31920.853,E2 31920.853} C_VEL
LIN {X 0,Y 731.704,Z 845.172,A -85,B 0,C 180,E1 31920.525,E2 31920.525} C_VEL
LIN {X 0,Y 731.92,Z 843.667,A -85,B 0,C 180,E1 31920.495,E2 31920.495} C_VEL
LIN {X 0,Y 734.577,Z 848.143,A -85,B 0,C 180,E1 31920.051,E2 31920.051} C_VEL
LIN {X 0,Y 735.379,Z 851.514,A -85,B 0,C 180,E1 31919.592,E2 31919.592} C_VEL
LIN {X 0,Y 734.594,Z 854.012,A -85,B 0,C 180,E1 31919.125,E2 31919.125} C_VEL
LIN {X 0,Y 732.334,Z 855.577,A -85,B 0,C 180,E1 31918.654,E2 31918.654} C_VEL
LIN {X 0,Y 728.594,Z 856.059,A -85,B 0,C 180,E1 31918.197,E2 31918.197} C_VEL
LIN {X 0,Y 724.115,Z 855.34,A -85,B 0,C 180,E1 31917.829,E2 31917.829} C_VEL
LIN {X 0,Y 713.847,Z 851.279,A -85,B 0,C 180,E1 31917.185,E2 31917.185} C_VEL
LIN {X 0,Y 704.127,Z 845.345,A -85,B 0,C 180,E1 31916.467,E2 31916.467} C_VEL
LIN {X 0,Y 695.845,Z 837.986,A -85,B 0,C 180,E1 31915.715,E2 31915.715} C_VEL
LIN {X 0,Y 688.882,Z 829.068,A -85,B 0,C 180,E1 31914.915,E2 31914.915} C_VEL
LIN {X 0,Y 683.629,Z 819.183,A -85,B 0,C 180,E1 31914.125,E2 31914.125} C_VEL
LIN {X 0,Y 679.698,Z 807.795,A -85,B 0,C 180,E1 31913.297,E2 31913.297} C_VEL
LIN {X 0,Y 676.95,Z 793.411,A -85,B 0,C 180,E1 31912.345,E2 31912.345} C_VEL
LIN {X 0,Y 675.725,Z 774.453,A -85,B 0,C 180,E1 31911.2,E2 31911.2} C_VEL
LIN {X 0,Y 677.909,Z 710.006,A -85,B 0,C 180,E1 31907.561,E2 31907.561} C_VEL
LIN {X 0,Y 678.948,Z 682.186,A -85,B 0,C 180,E1 31905.946,E2 31905.946} C_VEL
LIN {X 0,Y 667.995,Z 657.692,A -85,B 0,C 180,E1 31903.634,E2 31903.634} C_VEL
LIN {X 0,Y 664.802,Z 650.786,A -85,B 0,C 180,E1 31902.948,E2 31902.948} C_VEL
LIN {X 0,Y 664.631,Z 649.88,A -85,B 0,C 180,E1 31902.844,E2 31902.844} C_VEL
LIN {X 0,Y 664.637,Z 649.881,A -85,B 0,C 180,E1 31899.858,E2 31899.858} C_VEL
LIN {X 0,Y 664.644,Z 649.882,A -85,B 0,C 180,E1 31896.781,E2 31896.781} C_VEL
LIN {X 0,Y 664.64,Z 649.881,A -85,B 0,C 180,E1 31893.701,E2 31893.701} C_VEL
LIN {X 0,Y 664.644,Z 649.971,A -85,B 0,C 180,E1 31893.512,E2 31893.512} C_VEL
LIN {X 0,Y 671.198,Z 671.44,A -85,B 0,C 180,E1 31891.426,E2 31891.426} C_VEL
LIN {X 0,Y 670.61,Z 702.653,A -85,B 0,C 180,E1 31888.928,E2 31888.928} C_VEL
LIN {X 0,Y 674.045,Z 718.505,A -85,B 0,C 180,E1 31888.565,E2 31888.565} C_VEL
LIN {X 0,Y 672.515,Z 888.642,A -85,B 0,C 180,E1 31886.573,E2 31886.573} C_VEL
LIN {X 0,Y 671.754,Z 1003.159,A -85,B 0,C 180,E1 31885.276,E2 31885.276} C_VEL
LIN {X 0,Y 671.316,Z 1026.07,A -85,B 0,C 180,E1 31884.862,E2 31884.862} C_VEL
LIN {X 0,Y 670.848,Z 1046.813,A -85,B 0,C 180,E1 31884.338,E2 31884.338} C_VEL
LIN {X 0,Y 670.175,Z 1067.08,A -85,B 0,C 180,E1 31883.662,E2 31883.662} C_VEL
LIN {X 0,Y 669.407,Z 1087.642,A -85,B 0,C 180,E1 31882.811,E2 31882.811} C_VEL
LIN {X 0,Y 668.595,Z 1107.537,A -85,B 0,C 180,E1 31881.817,E2 31881.817} C_VEL
LIN {X 0,Y 667.798,Z 1126.444,A -85,B 0,C 180,E1 31880.693,E2 31880.693} C_VEL
LIN {X 0,Y 667,Z 1144.272,A -85,B 0,C 180,E1 31879.439,E2 31879.439} C_VEL
LIN {X 0,Y 666.254,Z 1161.175,A -85,B 0,C 180,E1 31878.054,E2 31878.054} C_VEL
LIN {X 0,Y 665.628,Z 1176.615,A -85,B 0,C 180,E1 31876.584,E2 31876.584} C_VEL
LIN {X 0,Y 665.098,Z 1190.984,A -85,B 0,C 180,E1 31874.986,E2 31874.986} C_VEL
LIN {X 0,Y 664.669,Z 1203.755,A -85,B 0,C 180,E1 31873.307,E2 31873.307} C_VEL
LIN {X 0,Y 664.35,Z 1215.132,A -85,B 0,C 180,E1 31871.536,E2 31871.536} C_VEL
LIN {X 0,Y 664.135,Z 1224.869,A -85,B 0,C 180,E1 31869.708,E2 31869.708} C_VEL
LIN {X 0,Y 664.016,Z 1232.747,A -85,B 0,C 180,E1 31867.876,E2 31867.876} C_VEL
LIN {X 0,Y 663.951,Z 1238.774,A -85,B 0,C 180,E1 31866.051,E2 31866.051} C_VEL
LIN {X 0,Y 663.913,Z 1243.378,A -85,B 0,C 180,E1 31864.146,E2 31864.146} C_VEL
LIN {X 0,Y 663.899,Z 1246.285,A -85,B 0,C 180,E1 31862.244,E2 31862.244} C_VEL
LIN {X 0,Y 663.909,Z 1247.384,A -85,B 0,C 180,E1 31860.431,E2 31860.431} C_VEL
LIN {X 0,Y 663.909,Z 1246.919,A -85,B 0,C 180,E1 31858.447,E2 31858.447} C_VEL
LIN {X 0,Y 663.907,Z 1244.812,A -85,B 0,C 180,E1 31856.546,E2 31856.546} C_VEL
LIN {X 0,Y 663.928,Z 1241.095,A -85,B 0,C 180,E1 31854.729,E2 31854.729} C_VEL
LIN {X 0,Y 663.982,Z 1235.525,A -85,B 0,C 180,E1 31852.82,E2 31852.82} C_VEL
LIN {X 0,Y 664.078,Z 1228.512,A -85,B 0,C 180,E1 31850.991,E2 31850.991} C_VEL
LIN {X 0,Y 664.237,Z 1219.999,A -85,B 0,C 180,E1 31849.242,E2 31849.242} C_VEL
LIN {X 0,Y 664.496,Z 1209.675,A -85,B 0,C 180,E1 31847.486,E2 31847.486} C_VEL
LIN {X 0,Y 664.857,Z 1197.998,A -85,B 0,C 180,E1 31845.81,E2 31845.81} C_VEL
LIN {X 0,Y 665.316,Z 1184.867,A -85,B 0,C 180,E1 31844.215,E2 31844.215} C_VEL
LIN {X 0,Y 665.874,Z 1170.33,A -85,B 0,C 180,E1 31842.703,E2 31842.703} C_VEL
LIN {X 0,Y 666.578,Z 1153.869,A -85,B 0,C 180,E1 31841.231,E2 31841.231} C_VEL
LIN {X 0,Y 667.335,Z 1137.013,A -85,B 0,C 180,E1 31839.933,E2 31839.933} C_VEL
LIN {X 0,Y 668.125,Z 1118.436,A -85,B 0,C 180,E1 31838.72,E2 31838.72} C_VEL
LIN {X 0,Y 668.925,Z 1099.792,A -85,B 0,C 180,E1 31837.687,E2 31837.687} C_VEL
LIN {X 0,Y 669.677,Z 1080.635,A -85,B 0,C 180,E1 31836.785,E2 31836.785} C_VEL
LIN {X 0,Y 670.411,Z 1060.713,A -85,B 0,C 180,E1 31836.02,E2 31836.02} C_VEL
LIN {X 0,Y 671.015,Z 1039.589,A -85,B 0,C 180,E1 31835.373,E2 31835.373} C_VEL
LIN {X 0,Y 671.545,Z 1017.733,A -85,B 0,C 180,E1 31834.869,E2 31834.869} C_VEL
LIN {X 0,Y 671.906,Z 995.69,A -85,B 0,C 180,E1 31834.519,E2 31834.519} C_VEL
LIN {X 0,Y 672.045,Z 978.015,A -85,B 0,C 180,E1 31834.316,E2 31834.316} C_VEL
LIN {X 0,Y 671.181,Z 970.423,A -85,B 0,C 180,E1 31834.197,E2 31834.197} C_VEL
LIN {X 0,Y 665.56,Z 950.585,A -85,B 0,C 180,E1 31833.754,E2 31833.754} C_VEL
LIN {X 0,Y 664.952,Z 944.057,A -85,B 0,C 180,E1 31833.654,E2 31833.654} C_VEL
LIN {X 0,Y 667.009,Z 718.963,A -85,B 0,C 180,E1 31831.02,E2 31831.02} C_VEL
LIN {X 0,Y 662.925,Z 700.933,A -85,B 0,C 180,E1 31830.581,E2 31830.581} C_VEL
LIN {X 0,Y 663.799,Z 673.972,A -85,B 0,C 180,E1 31828.329,E2 31828.329} C_VEL
LIN {X 0,Y 656.713,Z 650.872,A -85,B 0,C 180,E1 31825.923,E2 31825.923} C_VEL
LIN {X 0,Y 656.694,Z 650.868,A -85,B 0,C 180,E1 31822.781,E2 31822.781} C_VEL
LIN {X 0,Y 656.695,Z 650.866,A -85,B 0,C 180,E1 31819.715,E2 31819.715} C_VEL
LIN {X 0,Y 656.701,Z 650.869,A -85,B 0,C 180,E1 31816.631,E2 31816.631} C_VEL
LIN {X 0,Y 656.713,Z 650.867,A -85,B 0,C 180,E1 31813.489,E2 31813.489} C_VEL
LIN {X 0,Y 656.702,Z 650.864,A -85,B 0,C 180,E1 31810.421,E2 31810.421} C_VEL
LIN {X 0,Y 656.701,Z 650.862,A -85,B 0,C 180,E1 31807.301,E2 31807.301} C_VEL
LIN {X 0,Y 656.703,Z 650.867,A -85,B 0,C 180,E1 31804.184,E2 31804.184} C_VEL
LIN {X 0,Y 656.714,Z 650.864,A -85,B 0,C 180,E1 31801.075,E2 31801.075} C_VEL
LIN {X 0,Y 656.703,Z 650.862,A -85,B 0,C 180,E1 31797.968,E2 31797.968} C_VEL
LIN {X 0,Y 656.702,Z 650.864,A -85,B 0,C 180,E1 31794.842,E2 31794.842} C_VEL
LIN {X 0,Y 656.703,Z 650.869,A -85,B 0,C 180,E1 31791.716,E2 31791.716} C_VEL
LIN {X 0,Y 656.712,Z 650.863,A -85,B 0,C 180,E1 31788.648,E2 31788.648} C_VEL
LIN {X 0,Y 656.701,Z 650.863,A -85,B 0,C 180,E1 31785.454,E2 31785.454} C_VEL
LIN {X 0,Y 656.699,Z 650.861,A -85,B 0,C 180,E1 31782.309,E2 31782.309} C_VEL
LIN {X 0,Y 656.699,Z 650.864,A -85,B 0,C 180,E1 31779.201,E2 31779.201} C_VEL
LIN {X 0,Y 656.714,Z 650.865,A -85,B 0,C 180,E1 31776.119,E2 31776.119} C_VEL
LIN {X 0,Y 656.699,Z 650.861,A -85,B 0,C 180,E1 31772.969,E2 31772.969} C_VEL
LIN {X 0,Y 656.699,Z 650.86,A -85,B 0,C 180,E1 31769.827,E2 31769.827} C_VEL
LIN {X 0,Y 656.701,Z 650.866,A -85,B 0,C 180,E1 31766.772,E2 31766.772} C_VEL
LIN {X 0,Y 656.714,Z 650.866,A -85,B 0,C 180,E1 31763.62,E2 31763.62} C_VEL
LIN {X 0,Y 656.698,Z 650.864,A -85,B 0,C 180,E1 31760.448,E2 31760.448} C_VEL
LIN {X 0,Y 656.699,Z 650.864,A -85,B 0,C 180,E1 31757.336,E2 31757.336} C_VEL
LIN {X 0,Y 656.7,Z 650.868,A -85,B 0,C 180,E1 31754.215,E2 31754.215} C_VEL
LIN {X 0,Y 656.713,Z 650.867,A -85,B 0,C 180,E1 31751.078,E2 31751.078} C_VEL
LIN {X 0,Y 656.698,Z 650.865,A -85,B 0,C 180,E1 31747.91,E2 31747.91} C_VEL
LIN {X 0,Y 656.7,Z 650.862,A -85,B 0,C 180,E1 31744.863,E2 31744.863} C_VEL
LIN {X 0,Y 656.701,Z 650.868,A -85,B 0,C 180,E1 31741.738,E2 31741.738} C_VEL
LIN {X 0,Y 656.716,Z 650.868,A -85,B 0,C 180,E1 31738.622,E2 31738.622} C_VEL
LIN {X 0,Y 656.699,Z 650.867,A -85,B 0,C 180,E1 31735.46,E2 31735.46} C_VEL
LIN {X 0,Y 656.699,Z 650.867,A -85,B 0,C 180,E1 31732.35,E2 31732.35} C_VEL
LIN {X 0,Y 656.706,Z 650.868,A -85,B 0,C 180,E1 31729.31,E2 31729.31} C_VEL
LIN {X 0,Y 656.712,Z 650.867,A -85,B 0,C 180,E1 31726.153,E2 31726.153} C_VEL
LIN {X 0,Y 656.7,Z 650.869,A -85,B 0,C 180,E1 31723.01,E2 31723.01} C_VEL
LIN {X 0,Y 656.698,Z 650.942,A -85,B 0,C 180,E1 31722.709,E2 31722.709} C_VEL
LIN {X 0,Y 665.699,Z 676.943,A -85,B 0,C 180,E1 31720.205,E2 31720.205} C_VEL
LIN {X 0,Y 664.437,Z 716.282,A -85,B 0,C 180,E1 31717.334,E2 31717.334} C_VEL
LIN {X 0,Y 662.839,Z 761.695,A -85,B 0,C 180,E1 31714.093,E2 31714.093} C_VEL
LIN {X 0,Y 661.371,Z 807.678,A -85,B 0,C 180,E1 31710.863,E2 31710.863} C_VEL
LIN {X 0,Y 660.029,Z 855.097,A -85,B 0,C 180,E1 31707.573,E2 31707.573} C_VEL
LIN {X 0,Y 659.117,Z 895.898,A -85,B 0,C 180,E1 31704.802,E2 31704.802} C_VEL
LIN {X 0,Y 659.697,Z 902.805,A -85,B 0,C 180,E1 31704.696,E2 31704.696} C_VEL
LIN {X 0,Y 659.096,Z 970.279,A -85,B 0,C 180,E1 31703.889,E2 31703.889} C_VEL
LIN {X 0,Y 658.547,Z 1039.526,A -85,B 0,C 180,E1 31703.015,E2 31703.015} C_VEL
LIN {X 0,Y 658.365,Z 1056.67,A -85,B 0,C 180,E1 31702.62,E2 31702.62} C_VEL
LIN {X 0,Y 658.097,Z 1072.135,A -85,B 0,C 180,E1 31702.089,E2 31702.089} C_VEL
LIN {X 0,Y 657.787,Z 1086.722,A -85,B 0,C 180,E1 31701.422,E2 31701.422} C_VEL
LIN {X 0,Y 657.476,Z 1100.373,A -85,B 0,C 180,E1 31700.623,E2 31700.623} C_VEL
LIN {X 0,Y 657.142,Z 1113.645,A -85,B 0,C 180,E1 31699.641,E2 31699.641} C_VEL
LIN {X 0,Y 656.867,Z 1124.448,A -85,B 0,C 180,E1 31698.643,E2 31698.643} C_VEL
LIN {X 0,Y 656.614,Z 1134.06,A -85,B 0,C 180,E1 31697.549,E2 31697.549} C_VEL
LIN {X 0,Y 656.421,Z 1142.584,A -85,B 0,C 180,E1 31696.34,E2 31696.34} C_VEL
LIN {X 0,Y 656.278,Z 1149.875,A -85,B 0,C 180,E1 31695.003,E2 31695.003} C_VEL
LIN {X 0,Y 656.198,Z 1155.561,A -85,B 0,C 180,E1 31693.56,E2 31693.56} C_VEL
LIN {X 0,Y 656.161,Z 1159.018,A -85,B 0,C 180,E1 31692.229,E2 31692.229} C_VEL
LIN {X 0,Y 656.148,Z 1161.009,A -85,B 0,C 180,E1 31690.803,E2 31690.803} C_VEL
LIN {X 0,Y 656.15,Z 1161.289,A -85,B 0,C 180,E1 31689.384,E2 31689.384} C_VEL
LIN {X 0,Y 656.184,Z 1159.64,A -85,B 0,C 180,E1 31687.883,E2 31687.883} C_VEL
LIN {X 0,Y 656.24,Z 1156.313,A -85,B 0,C 180,E1 31686.474,E2 31686.474} C_VEL
LIN {X 0,Y 656.323,Z 1151.525,A -85,B 0,C 180,E1 31685.157,E2 31685.157} C_VEL
LIN {X 0,Y 656.489,Z 1144.466,A -85,B 0,C 180,E1 31683.755,E2 31683.755} C_VEL
LIN {X 0,Y 656.705,Z 1136.3,A -85,B 0,C 180,E1 31682.531,E2 31682.531} C_VEL
LIN {X 0,Y 656.986,Z 1126.795,A -85,B 0,C 180,E1 31681.395,E2 31681.395} C_VEL
LIN {X 0,Y 657.31,Z 1115.415,A -85,B 0,C 180,E1 31680.305,E2 31680.305} C_VEL
LIN {X 0,Y 657.677,Z 1102.25,A -85,B 0,C 180,E1 31679.303,E2 31679.303} C_VEL
LIN {X 0,Y 657.993,Z 1089.372,A -85,B 0,C 180,E1 31678.52,E2 31678.52} C_VEL
LIN {X 0,Y 658.339,Z 1074.655,A -85,B 0,C 180,E1 31677.824,E2 31677.824} C_VEL
LIN {X 0,Y 658.602,Z 1059.481,A -85,B 0,C 180,E1 31677.281,E2 31677.281} C_VEL
LIN {X 0,Y 658.76,Z 1043.272,A -85,B 0,C 180,E1 31676.884,E2 31676.884} C_VEL
LIN {X 0,Y 658.999,Z 1017.2,A -85,B 0,C 180,E1 31676.508,E2 31676.508} C_VEL
LIN {X 0,Y 660.544,Z 899.887,A -85,B 0,C 180,E1 31674.921,E2 31674.921} C_VEL
LIN {X 0,Y 662.309,Z 856.294,A -85,B 0,C 180,E1 31671.798,E2 31671.798} C_VEL
LIN {X 0,Y 664.643,Z 810.181,A -85,B 0,C 180,E1 31668.414,E2 31668.414} C_VEL
LIN {X 0,Y 667.512,Z 765.499,A -85,B 0,C 180,E1 31665.046,E2 31665.046} C_VEL
LIN {X 0,Y 670.919,Z 722.79,A -85,B 0,C 180,E1 31661.717,E2 31661.717} C_VEL
LIN {X 0,Y 673.325,Z 689.071,A -85,B 0,C 180,E1 31658.916,E2 31658.916} C_VEL
LIN {X 0,Y 667.813,Z 675.056,A -85,B 0,C 180,E1 31656.996,E2 31656.996} C_VEL
LIN {X 0,Y 662.886,Z 663.896,A -85,B 0,C 180,E1 31655.232,E2 31655.232} C_VEL
LIN {X 0,Y 660.663,Z 659.375,A -85,B 0,C 180,E1 31654.421,E2 31654.421} C_VEL
LIN {X 0,Y 658.57,Z 655.087,A -85,B 0,C 180,E1 31653.604,E2 31653.604} C_VEL
LIN {X 0,Y 656.885,Z 651.887,A -85,B 0,C 180,E1 31652.927,E2 31652.927} C_VEL
LIN {X 0,Y 656.693,Z 650.87,A -85,B 0,C 180,E1 31652.722,E2 31652.722} C_VEL
LIN {X 0,Y 656.69,Z 650.87,A -85,B 0,C 180,E1 31649.688,E2 31649.688} C_VEL
LIN {X 0,Y 656.691,Z 650.871,A -85,B 0,C 180,E1 31646.656,E2 31646.656} C_VEL
LIN {X 0,Y 656.69,Z 650.871,A -85,B 0,C 180,E1 31643.652,E2 31643.652} C_VEL
LIN {X 0,Y 656.695,Z 650.868,A -85,B 0,C 180,E1 31640.665,E2 31640.665} C_VEL
LIN {X 0,Y 656.729,Z 651.107,A -85,B 0,C 180,E1 31638.291,E2 31638.291} C_VEL
LIN {X 0,Y 658.247,Z 654.69,A -85,B 0,C 180,E1 31637.706,E2 31637.706} C_VEL
LIN {X 0,Y 659.291,Z 656.085,A -85,B 0,C 180,E1 31637.436,E2 31637.436} C_VEL
LIN {X 0,Y 661.061,Z 659.792,A -85,B 0,C 180,E1 31636.868,E2 31636.868} C_VEL
LIN {X 0,Y 665.655,Z 669.3,A -85,B 0,C 180,E1 31635.574,E2 31635.574} C_VEL
LIN {X 0,Y 670.618,Z 680.892,A -85,B 0,C 180,E1 31634.247,E2 31634.247} C_VEL
LIN {X 0,Y 671.592,Z 683.496,A -85,B 0,C 180,E1 31633.98,E2 31633.98} C_VEL
LIN {X 0,Y 668.09,Z 727.574,A -85,B 0,C 180,E1 31631.356,E2 31631.356} C_VEL
LIN {X 0,Y 666.088,Z 771.457,A -85,B 0,C 180,E1 31628.862,E2 31628.862} C_VEL
LIN {X 0,Y 667.207,Z 791.055,A -85,B 0,C 180,E1 31627.691,E2 31627.691} C_VEL
LIN {X 0,Y 669.713,Z 805.421,A -85,B 0,C 180,E1 31626.775,E2 31626.775} C_VEL
LIN {X 0,Y 673.595,Z 817.802,A -85,B 0,C 180,E1 31625.929,E2 31625.929} C_VEL
LIN {X 0,Y 679.314,Z 829.451,A -85,B 0,C 180,E1 31625.076,E2 31625.076} C_VEL
LIN {X 0,Y 686.299,Z 839.217,A -85,B 0,C 180,E1 31624.301,E2 31624.301} C_VEL
LIN {X 0,Y 694.803,Z 847.685,A -85,B 0,C 180,E1 31623.567,E2 31623.567} C_VEL
LIN {X 0,Y 704.8,Z 854.862,A -85,B 0,C 180,E1 31622.874,E2 31622.874} C_VEL
LIN {X 0,Y 715.875,Z 860.439,A -85,B 0,C 180,E1 31622.244,E2 31622.244} C_VEL
LIN {X 0,Y 722.008,Z 862.547,A -85,B 0,C 180,E1 31621.904,E2 31621.904} C_VEL
LIN {X 0,Y 726.734,Z 863.177,A -85,B 0,C 180,E1 31621.52,E2 31621.52} C_VEL
LIN {X 0,Y 730.445,Z 862.576,A -85,B 0,C 180,E1 31621.067,E2 31621.067} C_VEL
LIN {X 0,Y 732.674,Z 860.95,A -85,B 0,C 180,E1 31620.598,E2 31620.598} C_VEL
LIN {X 0,Y 733.431,Z 858.284,A -85,B 0,C 180,E1 31620.11,E2 31620.11} C_VEL
LIN {X 0,Y 733.215,Z 857.18,A -85,B 0,C 180,E1 31619.914,E2 31619.914} C_VEL
LIN {X 0,Y 728.507,Z 876.954,A -85,B 0,C 180,E1 31619.643,E2 31619.643} C_VEL
LIN {X 0,Y 725.884,Z 886.402,A -85,B 0,C 180,E1 31619.459,E2 31619.459} C_VEL
LIN {X 0,Y 719.659,Z 904.029,A -85,B 0,C 180,E1 31619.359,E2 31619.359} C_VEL
LIN {X 0,Y 711.71,Z 921.269,A -85,B 0,C 180,E1 31619.2,E2 31619.2} C_VEL
LIN {X 0,Y 702.441,Z 937.846,A -85,B 0,C 180,E1 31618.943,E2 31618.943} C_VEL
LIN {X 0,Y 692.535,Z 953.923,A -85,B 0,C 180,E1 31618.547,E2 31618.547} C_VEL
LIN {X 0,Y 683.847,Z 969.589,A -85,B 0,C 180,E1 31618.038,E2 31618.038} C_VEL
LIN {X 0,Y 678.437,Z 982.48,A -85,B 0,C 180,E1 31617.565,E2 31617.565} C_VEL
LIN {X 0,Y 676.679,Z 986.79,A -85,B 0,C 180,E1 31617.404,E2 31617.404} C_VEL
LIN {X 0,Y 671.353,Z 998.697,A -85,B 0,C 180,E1 31616.967,E2 31616.967} C_VEL
LIN {X 0,Y 665.405,Z 1018.258,A -85,B 0,C 180,E1 31616.168,E2 31616.168} C_VEL
LIN {X 0,Y 664.399,Z 1023.165,A -85,B 0,C 180,E1 31615.983,E2 31615.983} C_VEL
LIN {X 0,Y 664.052,Z 1064.401,A -85,B 0,C 180,E1 31615.5,E2 31615.5} C_VEL
LIN {X 0,Y 663.596,Z 1088.003,A -85,B 0,C 180,E1 31615.059,E2 31615.059} C_VEL
LIN {X 0,Y 663.064,Z 1110.473,A -85,B 0,C 180,E1 31614.475,E2 31614.475} C_VEL
LIN {X 0,Y 662.433,Z 1131.578,A -85,B 0,C 180,E1 31613.765,E2 31613.765} C_VEL
LIN {X 0,Y 661.739,Z 1151.958,A -85,B 0,C 180,E1 31612.916,E2 31612.916} C_VEL
LIN {X 0,Y 661.002,Z 1169.215,A -85,B 0,C 180,E1 31612.032,E2 31612.032} C_VEL
LIN {X 0,Y 660.088,Z 1188.463,A -85,B 0,C 180,E1 31610.852,E2 31610.852} C_VEL
LIN {X 0,Y 659.264,Z 1205.357,A -85,B 0,C 180,E1 31609.634,E2 31609.634} C_VEL
LIN {X 0,Y 658.578,Z 1219.62,A -85,B 0,C 180,E1 31608.453,E2 31608.453} C_VEL
LIN {X 0,Y 657.955,Z 1233.521,A -85,B 0,C 180,E1 31607.145,E2 31607.145} C_VEL
LIN {X 0,Y 657.325,Z 1248.333,A -85,B 0,C 180,E1 31605.527,E2 31605.527} C_VEL
LIN {X 0,Y 656.864,Z 1260.235,A -85,B 0,C 180,E1 31604.005,E2 31604.005} C_VEL
LIN {X 0,Y 656.535,Z 1270.516,A -85,B 0,C 180,E1 31602.488,E2 31602.488} C_VEL
LIN {X 0,Y 656.23,Z 1281.605,A -85,B 0,C 180,E1 31600.534,E2 31600.534} C_VEL
LIN {X 0,Y 656.07,Z 1289.373,A -85,B 0,C 180,E1 31598.853,E2 31598.853} C_VEL
LIN {X 0,Y 655.978,Z 1295.992,A -85,B 0,C 180,E1 31597.091,E2 31597.091} C_VEL
LIN {X 0,Y 655.933,Z 1301.411,A -85,B 0,C 180,E1 31595.159,E2 31595.159} C_VEL
LIN {X 0,Y 655.919,Z 1304.81,A -85,B 0,C 180,E1 31593.407,E2 31593.407} C_VEL
LIN {X 0,Y 655.907,Z 1306.915,A -85,B 0,C 180,E1 31591.571,E2 31591.571} C_VEL
LIN {X 0,Y 655.9,Z 1307.39,A -85,B 0,C 180,E1 31589.562,E2 31589.562} C_VEL
LIN {X 0,Y 655.909,Z 1306.435,A -85,B 0,C 180,E1 31587.902,E2 31587.902} C_VEL
LIN {X 0,Y 655.911,Z 1303.974,A -85,B 0,C 180,E1 31586.065,E2 31586.065} C_VEL
LIN {X 0,Y 655.933,Z 1299.385,A -85,B 0,C 180,E1 31584.049,E2 31584.049} C_VEL
LIN {X 0,Y 655.999,Z 1294.128,A -85,B 0,C 180,E1 31582.379,E2 31582.379} C_VEL
LIN {X 0,Y 656.133,Z 1286.741,A -85,B 0,C 180,E1 31580.526,E2 31580.526} C_VEL
LIN {X 0,Y 656.333,Z 1277.326,A -85,B 0,C 180,E1 31578.665,E2 31578.665} C_VEL
LIN {X 0,Y 656.595,Z 1268.195,A -85,B 0,C 180,E1 31577.153,E2 31577.153} C_VEL
LIN {X 0,Y 656.997,Z 1256.953,A -85,B 0,C 180,E1 31575.546,E2 31575.546} C_VEL
LIN {X 0,Y 657.548,Z 1242.813,A -85,B 0,C 180,E1 31573.842,E2 31573.842} C_VEL
LIN {X 0,Y 658.103,Z 1229.819,A -85,B 0,C 180,E1 31572.491,E2 31572.491} C_VEL
LIN {X 0,Y 658.84,Z 1214.457,A -85,B 0,C 180,E1 31571.093,E2 31571.093} C_VEL
LIN {X 0,Y 659.747,Z 1195.694,A -85,B 0,C 180,E1 31569.645,E2 31569.645} C_VEL
LIN {X 0,Y 660.644,Z 1177.012,A -85,B 0,C 180,E1 31568.42,E2 31568.42} C_VEL
LIN {X 0,Y 661.498,Z 1158.35,A -85,B 0,C 180,E1 31567.389,E2 31567.389} C_VEL
LIN {X 0,Y 662.216,Z 1138.747,A -85,B 0,C 180,E1 31566.507,E2 31566.507} C_VEL
LIN {X 0,Y 662.929,Z 1116.929,A -85,B 0,C 180,E1 31565.707,E2 31565.707} C_VEL
LIN {X 0,Y 663.591,Z 1094.3,A -85,B 0,C 180,E1 31565.058,E2 31565.058} C_VEL
LIN {X 0,Y 664.076,Z 1071.326,A -85,B 0,C 180,E1 31564.57,E2 31564.57} C_VEL
LIN {X 0,Y 664.432,Z 1046.762,A -85,B 0,C 180,E1 31564.23,E2 31564.23} C_VEL
LIN {X 0,Y 664.729,Z 1022.404,A -85,B 0,C 180,E1 31563.944,E2 31563.944} C_VEL
LIN {X 0,Y 668.158,Z 1009.892,A -85,B 0,C 180,E1 31563.419,E2 31563.419} C_VEL
LIN {X 0,Y 672.514,Z 996.584,A -85,B 0,C 180,E1 31562.889,E2 31562.889} C_VEL
LIN {X 0,Y 678.34,Z 983.479,A -85,B 0,C 180,E1 31562.428,E2 31562.428} C_VEL
LIN {X 0,Y 683.307,Z 971.139,A -85,B 0,C 180,E1 31561.983,E2 31561.983} C_VEL
LIN {X 0,Y 691.873,Z 955.091,A -85,B 0,C 180,E1 31561.484,E2 31561.484} C_VEL
LIN {X 0,Y 701.811,Z 938.884,A -85,B 0,C 180,E1 31561.077,E2 31561.077} C_VEL
LIN {X 0,Y 711.389,Z 921.896,A -85,B 0,C 180,E1 31560.808,E2 31560.808} C_VEL
LIN {X 0,Y 719.276,Z 904.963,A -85,B 0,C 180,E1 31560.647,E2 31560.647} C_VEL
LIN {X 0,Y 725.753,Z 886.84,A -85,B 0,C 180,E1 31560.543,E2 31560.543} C_VEL
LIN {X 0,Y 726.964,Z 882.589,A -85,B 0,C 180,E1 31560.472,E2 31560.472} C_VEL
LIN {X 0,Y 731.126,Z 866.673,A -85,B 0,C 180,E1 31560.201,E2 31560.201} C_VEL
LIN {X 0,Y 733.26,Z 856.972,A -85,B 0,C 180,E1 31560.082,E2 31560.082} C_VEL
LIN {X 0,Y 733.183,Z 859.963,A -85,B 0,C 180,E1 31559.604,E2 31559.604} C_VEL
LIN {X 0,Y 731.566,Z 862.008,A -85,B 0,C 180,E1 31559.131,E2 31559.131} C_VEL
LIN {X 0,Y 728.898,Z 863.003,A -85,B 0,C 180,E1 31558.718,E2 31558.718} C_VEL
LIN {X 0,Y 724.969,Z 863.074,A -85,B 0,C 180,E1 31558.319,E2 31558.319} C_VEL
LIN {X 0,Y 719.621,Z 861.869,A -85,B 0,C 180,E1 31557.949,E2 31557.949} C_VEL
LIN {X 0,Y 708.489,Z 857.257,A -85,B 0,C 180,E1 31557.261,E2 31557.261} C_VEL
LIN {X 0,Y 698.783,Z 851.241,A -85,B 0,C 180,E1 31556.535,E2 31556.535} C_VEL
LIN {X 0,Y 690.481,Z 843.946,A -85,B 0,C 180,E1 31555.779,E2 31555.779} C_VEL
LIN {X 0,Y 683.571,Z 835.453,A -85,B 0,C 180,E1 31554.999,E2 31554.999} C_VEL
LIN {X 0,Y 678.033,Z 825.788,A -85,B 0,C 180,E1 31554.202,E2 31554.202} C_VEL
LIN {X 0,Y 673.46,Z 813.71,A -85,B 0,C 180,E1 31553.297,E2 31553.297} C_VEL
LIN {X 0,Y 670.459,Z 800.022,A -85,B 0,C 180,E1 31552.365,E2 31552.365} C_VEL
LIN {X 0,Y 668.843,Z 781.524,A -85,B 0,C 180,E1 31551.215,E2 31551.215} C_VEL
LIN {X 0,Y 669.313,Z 753.927,A -85,B 0,C 180,E1 31549.632,E2 31549.632} C_VEL
LIN {X 0,Y 671.437,Z 705.739,A -85,B 0,C 180,E1 31546.879,E2 31546.879} C_VEL
LIN {X 0,Y 672.247,Z 685.891,A -85,B 0,C 180,E1 31545.712,E2 31545.712} C_VEL
LIN {X 0,Y 661.591,Z 662.151,A -85,B 0,C 180,E1 31543.446,E2 31543.446} C_VEL
LIN {X 0,Y 656.853,Z 651.741,A -85,B 0,C 180,E1 31542.404,E2 31542.404} C_VEL
LIN {X 0,Y 656.701,Z 650.87,A -85,B 0,C 180,E1 31542.298,E2 31542.298} C_VEL
LIN {X 0,Y 656.714,Z 650.866,A -85,B 0,C 180,E1 31539.188,E2 31539.188} C_VEL
LIN {X 0,Y 656.703,Z 650.869,A -85,B 0,C 180,E1 31535.996,E2 31535.996} C_VEL
LIN {X 0,Y 656.716,Z 650.949,A -85,B 0,C 180,E1 31533.922,E2 31533.922} C_VEL
LIN {X 0,Y 662.534,Z 669.378,A -85,B 0,C 180,E1 31532.089,E2 31532.089} C_VEL
LIN {X 0,Y 663.971,Z 675.245,A -85,B 0,C 180,E1 31531.531,E2 31531.531} C_VEL
LIN {X 0,Y 663.399,Z 703.331,A -85,B 0,C 180,E1 31529.272,E2 31529.272} C_VEL
LIN {X 0,Y 666.962,Z 719.987,A -85,B 0,C 180,E1 31528.87,E2 31528.87} C_VEL
LIN {X 0,Y 665.183,Z 884.705,A -85,B 0,C 180,E1 31526.89,E2 31526.89} C_VEL
LIN {X 0,Y 664.27,Z 1003.998,A -85,B 0,C 180,E1 31525.511,E2 31525.511} C_VEL
LIN {X 0,Y 663.811,Z 1026.823,A -85,B 0,C 180,E1 31525.092,E2 31525.092} C_VEL
LIN {X 0,Y 663.291,Z 1048.275,A -85,B 0,C 180,E1 31524.539,E2 31524.539} C_VEL
LIN {X 0,Y 662.625,Z 1068.768,A -85,B 0,C 180,E1 31523.854,E2 31523.854} C_VEL
LIN {X 0,Y 661.879,Z 1088.478,A -85,B 0,C 180,E1 31523.033,E2 31523.033} C_VEL
LIN {X 0,Y 661.07,Z 1107.546,A -85,B 0,C 180,E1 31522.078,E2 31522.078} C_VEL
LIN {X 0,Y 660.201,Z 1126.452,A -85,B 0,C 180,E1 31520.942,E2 31520.942} C_VEL
LIN {X 0,Y 659.321,Z 1144.278,A -85,B 0,C 180,E1 31519.674,E2 31519.674} C_VEL
LIN {X 0,Y 658.499,Z 1161.333,A -85,B 0,C 180,E1 31518.26,E2 31518.26} C_VEL
LIN {X 0,Y 657.821,Z 1176.62,A -85,B 0,C 180,E1 31516.786,E2 31516.786} C_VEL
LIN {X 0,Y 657.228,Z 1190.986,A -85,B 0,C 180,E1 31515.17,E2 31515.17} C_VEL
LIN {X 0,Y 656.773,Z 1203.126,A -85,B 0,C 180,E1 31513.56,E2 31513.56} C_VEL
LIN {X 0,Y 656.412,Z 1214.554,A -85,B 0,C 180,E1 31511.778,E2 31511.778} C_VEL
LIN {X 0,Y 656.189,Z 1224.06,A -85,B 0,C 180,E1 31510.004,E2 31510.004} C_VEL
LIN {X 0,Y 656.038,Z 1232.047,A -85,B 0,C 180,E1 31508.149,E2 31508.149} C_VEL
LIN {X 0,Y 655.958,Z 1238.271,A -85,B 0,C 180,E1 31506.301,E2 31506.301} C_VEL
LIN {X 0,Y 655.925,Z 1242.902,A -85,B 0,C 180,E1 31504.459,E2 31504.459} C_VEL
LIN {X 0,Y 655.911,Z 1245.839,A -85,B 0,C 180,E1 31502.621,E2 31502.621} C_VEL
LIN {X 0,Y 655.911,Z 1247.338,A -85,B 0,C 180,E1 31500.611,E2 31500.611} C_VEL
LIN {X 0,Y 655.902,Z 1247.184,A -85,B 0,C 180,E1 31498.777,E2 31498.777} C_VEL
LIN {X 0,Y 655.901,Z 1245.317,A -85,B 0,C 180,E1 31496.883,E2 31496.883} C_VEL
LIN {X 0,Y 655.926,Z 1241.711,A -85,B 0,C 180,E1 31494.928,E2 31494.928} C_VEL
LIN {X 0,Y 655.979,Z 1236.729,A -85,B 0,C 180,E1 31493.084,E2 31493.084} C_VEL
LIN {X 0,Y 656.062,Z 1229.946,A -85,B 0,C 180,E1 31491.233,E2 31491.233} C_VEL
LIN {X 0,Y 656.241,Z 1221.219,A -85,B 0,C 180,E1 31489.347,E2 31489.347} C_VEL
LIN {X 0,Y 656.513,Z 1211.38,A -85,B 0,C 180,E1 31487.599,E2 31487.599} C_VEL
LIN {X 0,Y 656.887,Z 1199.967,A -85,B 0,C 180,E1 31485.904,E2 31485.904} C_VEL
LIN {X 0,Y 657.37,Z 1187.16,A -85,B 0,C 180,E1 31484.291,E2 31484.291} C_VEL
LIN {X 0,Y 658.01,Z 1172.162,A -85,B 0,C 180,E1 31482.672,E2 31482.672} C_VEL
LIN {X 0,Y 658.752,Z 1156.61,A -85,B 0,C 180,E1 31481.229,E2 31481.229} C_VEL
LIN {X 0,Y 659.556,Z 1139.431,A -85,B 0,C 180,E1 31479.871,E2 31479.871} C_VEL
LIN {X 0,Y 660.421,Z 1121.258,A -85,B 0,C 180,E1 31478.642,E2 31478.642} C_VEL
LIN {X 0,Y 661.318,Z 1102.423,A -85,B 0,C 180,E1 31477.556,E2 31477.556} C_VEL
LIN {X 0,Y 662.14,Z 1082.508,A -85,B 0,C 180,E1 31476.6,E2 31476.6} C_VEL
LIN {X 0,Y 662.894,Z 1062.656,A -85,B 0,C 180,E1 31475.825,E2 31475.825} C_VEL
LIN {X 0,Y 663.58,Z 1040.397,A -85,B 0,C 180,E1 31475.129,E2 31475.129} C_VEL
LIN {X 0,Y 664.151,Z 1018.552,A -85,B 0,C 180,E1 31474.615,E2 31474.615} C_VEL
LIN {X 0,Y 664.538,Z 996.501,A -85,B 0,C 180,E1 31474.258,E2 31474.258} C_VEL
LIN {X 0,Y 664.952,Z 944.057,A -85,B 0,C 180,E1 31473.654,E2 31473.654} C_VEL
LIN {X 0,Y 664.141,Z 936.465,A -85,B 0,C 180,E1 31473.534,E2 31473.534} C_VEL
LIN {X 0,Y 658.615,Z 916.636,A -85,B 0,C 180,E1 31473.075,E2 31473.075} C_VEL
LIN {X 0,Y 657.978,Z 910.113,A -85,B 0,C 180,E1 31472.971,E2 31472.971} C_VEL
LIN {X 0,Y 659.979,Z 720.375,A -85,B 0,C 180,E1 31470.699,E2 31470.699} C_VEL
LIN {X 0,Y 655.639,Z 701.201,A -85,B 0,C 180,E1 31470.223,E2 31470.223} C_VEL
LIN {X 0,Y 656.387,Z 676.497,A -85,B 0,C 180,E1 31468.141,E2 31468.141} C_VEL
LIN {X 0,Y 649.522,Z 654.379,A -85,B 0,C 180,E1 31465.837,E2 31465.837} C_VEL
LIN {X 0,Y 648.762,Z 651.862,A -85,B 0,C 180,E1 31465.544,E2 31465.544} C_VEL
LIN {X 0,Y 648.751,Z 651.859,A -85,B 0,C 180,E1 31462.497,E2 31462.497} C_VEL
LIN {X 0,Y 648.75,Z 651.856,A -85,B 0,C 180,E1 31459.451,E2 31459.451} C_VEL
LIN {X 0,Y 648.753,Z 651.858,A -85,B 0,C 180,E1 31456.419,E2 31456.419} C_VEL
LIN {X 0,Y 648.771,Z 651.86,A -85,B 0,C 180,E1 31453.302,E2 31453.302} C_VEL
LIN {X 0,Y 648.753,Z 651.855,A -85,B 0,C 180,E1 31450.225,E2 31450.225} C_VEL
LIN {X 0,Y 648.755,Z 651.851,A -85,B 0,C 180,E1 31447.17,E2 31447.17} C_VEL
LIN {X 0,Y 648.761,Z 651.856,A -85,B 0,C 180,E1 31444.126,E2 31444.126} C_VEL
LIN {X 0,Y 648.775,Z 651.854,A -85,B 0,C 180,E1 31440.982,E2 31440.982} C_VEL
LIN {X 0,Y 648.757,Z 651.852,A -85,B 0,C 180,E1 31437.84,E2 31437.84} C_VEL
LIN {X 0,Y 648.76,Z 651.853,A -85,B 0,C 180,E1 31434.786,E2 31434.786} C_VEL
LIN {X 0,Y 648.761,Z 651.858,A -85,B 0,C 180,E1 31431.664,E2 31431.664} C_VEL
LIN {X 0,Y 648.773,Z 651.854,A -85,B 0,C 180,E1 31428.512,E2 31428.512} C_VEL
LIN {X 0,Y 648.757,Z 651.853,A -85,B 0,C 180,E1 31425.373,E2 31425.373} C_VEL
LIN {X 0,Y 648.758,Z 651.85,A -85,B 0,C 180,E1 31422.272,E2 31422.272} C_VEL
LIN {X 0,Y 648.762,Z 651.853,A -85,B 0,C 180,E1 31419.225,E2 31419.225} C_VEL
LIN {X 0,Y 648.775,Z 651.854,A -85,B 0,C 180,E1 31416.106,E2 31416.106} C_VEL
LIN {X 0,Y 648.758,Z 651.851,A -85,B 0,C 180,E1 31412.89,E2 31412.89} C_VEL
LIN {X 0,Y 648.76,Z 651.849,A -85,B 0,C 180,E1 31409.825,E2 31409.825} C_VEL
LIN {X 0,Y 648.76,Z 651.854,A -85,B 0,C 180,E1 31406.732,E2 31406.732} C_VEL
LIN {X 0,Y 648.775,Z 651.854,A -85,B 0,C 180,E1 31403.63,E2 31403.63} C_VEL
LIN {X 0,Y 648.762,Z 651.852,A -85,B 0,C 180,E1 31400.509,E2 31400.509} C_VEL
LIN {X 0,Y 648.759,Z 651.853,A -85,B 0,C 180,E1 31397.319,E2 31397.319} C_VEL
LIN {X 0,Y 648.765,Z 651.858,A -85,B 0,C 180,E1 31394.263,E2 31394.263} C_VEL
LIN {X 0,Y 648.774,Z 651.856,A -85,B 0,C 180,E1 31391.118,E2 31391.118} C_VEL
LIN {X 0,Y 648.759,Z 651.854,A -85,B 0,C 180,E1 31387.912,E2 31387.912} C_VEL
LIN {X 0,Y 648.758,Z 651.851,A -85,B 0,C 180,E1 31384.785,E2 31384.785} C_VEL
LIN {X 0,Y 648.764,Z 651.858,A -85,B 0,C 180,E1 31381.763,E2 31381.763} C_VEL
LIN {X 0,Y 648.776,Z 651.856,A -85,B 0,C 180,E1 31378.608,E2 31378.608} C_VEL
LIN {X 0,Y 648.759,Z 651.856,A -85,B 0,C 180,E1 31375.449,E2 31375.449} C_VEL
LIN {X 0,Y 648.764,Z 651.856,A -85,B 0,C 180,E1 31372.389,E2 31372.389} C_VEL
LIN {X 0,Y 648.768,Z 651.857,A -85,B 0,C 180,E1 31369.313,E2 31369.313} C_VEL
LIN {X 0,Y 648.774,Z 651.856,A -85,B 0,C 180,E1 31366.161,E2 31366.161} C_VEL
LIN {X 0,Y 648.781,Z 651.98,A -85,B 0,C 180,E1 31363.117,E2 31363.117} C_VEL
LIN {X 0,Y 658.26,Z 679.24,A -85,B 0,C 180,E1 31360.449,E2 31360.449} C_VEL
LIN {X 0,Y 658.407,Z 683.19,A -85,B 0,C 180,E1 31360.141,E2 31360.141} C_VEL
LIN {X 0,Y 657.033,Z 721.512,A -85,B 0,C 180,E1 31357.333,E2 31357.333} C_VEL
LIN {X 0,Y 655.417,Z 764.72,A -85,B 0,C 180,E1 31354.226,E2 31354.226} C_VEL
LIN {X 0,Y 653.867,Z 809.913,A -85,B 0,C 180,E1 31351.02,E2 31351.02} C_VEL
LIN {X 0,Y 652.426,Z 858.163,A -85,B 0,C 180,E1 31347.651,E2 31347.651} C_VEL
LIN {X 0,Y 651.496,Z 896.436,A -85,B 0,C 180,E1 31345.027,E2 31345.027} C_VEL
LIN {X 0,Y 652.127,Z 903.406,A -85,B 0,C 180,E1 31344.918,E2 31344.918} C_VEL
LIN {X 0,Y 650.828,Z 1039.664,A -85,B 0,C 180,E1 31343.199,E2 31343.199} C_VEL
LIN {X 0,Y 650.637,Z 1056.641,A -85,B 0,C 180,E1 31342.809,E2 31342.809} C_VEL
LIN {X 0,Y 650.383,Z 1071.215,A -85,B 0,C 180,E1 31342.317,E2 31342.317} C_VEL
LIN {X 0,Y 650.056,Z 1085.716,A -85,B 0,C 180,E1 31341.664,E2 31341.664} C_VEL
LIN {X 0,Y 649.712,Z 1099.495,A -85,B 0,C 180,E1 31340.872,E2 31340.872} C_VEL
LIN {X 0,Y 649.37,Z 1112.305,A -85,B 0,C 180,E1 31339.942,E2 31339.942} C_VEL
LIN {X 0,Y 649.041,Z 1124.118,A -85,B 0,C 180,E1 31338.876,E2 31338.876} C_VEL
LIN {X 0,Y 648.752,Z 1134.202,A -85,B 0,C 180,E1 31337.739,E2 31337.739} C_VEL
LIN {X 0,Y 648.524,Z 1143.14,A -85,B 0,C 180,E1 31336.472,E2 31336.472} C_VEL
LIN {X 0,Y 648.374,Z 1150.159,A -85,B 0,C 180,E1 31335.199,E2 31335.199} C_VEL
LIN {X 0,Y 648.263,Z 1156.274,A -85,B 0,C 180,E1 31333.668,E2 31333.668} C_VEL
LIN {X 0,Y 648.222,Z 1159.894,A -85,B 0,C 180,E1 31332.29,E2 31332.29} C_VEL
LIN {X 0,Y 648.206,Z 1161.926,A -85,B 0,C 180,E1 31330.847,E2 31330.847} C_VEL
LIN {X 0,Y 648.208,Z 1162.259,A -85,B 0,C 180,E1 31329.411,E2 31329.411} C_VEL
LIN {X 0,Y 648.246,Z 1160.669,A -85,B 0,C 180,E1 31327.89,E2 31327.89} C_VEL
LIN {X 0,Y 648.316,Z 1157.426,A -85,B 0,C 180,E1 31326.465,E2 31326.465} C_VEL
LIN {X 0,Y 648.415,Z 1152.299,A -85,B 0,C 180,E1 31325.043,E2 31325.043} C_VEL
LIN {X 0,Y 648.594,Z 1145.682,A -85,B 0,C 180,E1 31323.712,E2 31323.712} C_VEL
LIN {X 0,Y 648.836,Z 1137.623,A -85,B 0,C 180,E1 31322.473,E2 31322.473} C_VEL
LIN {X 0,Y 649.172,Z 1127.406,A -85,B 0,C 180,E1 31321.236,E2 31321.236} C_VEL
LIN {X 0,Y 649.514,Z 1116.46,A -85,B 0,C 180,E1 31320.176,E2 31320.176} C_VEL
LIN {X 0,Y 649.917,Z 1103.35,A -85,B 0,C 180,E1 31319.163,E2 31319.163} C_VEL
LIN {X 0,Y 650.261,Z 1090.537,A -85,B 0,C 180,E1 31318.37,E2 31318.37} C_VEL
LIN {X 0,Y 650.632,Z 1075.912,A -85,B 0,C 180,E1 31317.666,E2 31317.666} C_VEL
LIN {X 0,Y 650.916,Z 1060.925,A -85,B 0,C 180,E1 31317.116,E2 31317.116} C_VEL
LIN {X 0,Y 651.085,Z 1044.938,A -85,B 0,C 180,E1 31316.712,E2 31316.712} C_VEL
LIN {X 0,Y 651.321,Z 1020.534,A -85,B 0,C 180,E1 31316.342,E2 31316.342} C_VEL
LIN {X 0,Y 653.193,Z 901.102,A -85,B 0,C 180,E1 31314.659,E2 31314.659} C_VEL
LIN {X 0,Y 655.133,Z 857.276,A -85,B 0,C 180,E1 31311.481,E2 31311.481} C_VEL
LIN {X 0,Y 657.628,Z 811.917,A -85,B 0,C 180,E1 31308.111,E2 31308.111} C_VEL
LIN {X 0,Y 660.764,Z 767.149,A -85,B 0,C 180,E1 31304.689,E2 31304.689} C_VEL
LIN {X 0,Y 664.406,Z 724.881,A -85,B 0,C 180,E1 31301.349,E2 31301.349} C_VEL
LIN {X 0,Y 666.953,Z 693.257,A -85,B 0,C 180,E1 31298.681,E2 31298.681} C_VEL
LIN {X 0,Y 661.815,Z 680.018,A -85,B 0,C 180,E1 31296.823,E2 31296.823} C_VEL
LIN {X 0,Y 657.453,Z 669.741,A -85,B 0,C 180,E1 31295.181,E2 31295.181} C_VEL
LIN {X 0,Y 654.816,Z 664.53,A -85,B 0,C 180,E1 31294.203,E2 31294.203} C_VEL
LIN {X 0,Y 652.974,Z 660.646,A -85,B 0,C 180,E1 31293.44,E2 31293.44} C_VEL
LIN {X 0,Y 651.337,Z 656.949,A -85,B 0,C 180,E1 31292.677,E2 31292.677} C_VEL
LIN {X 0,Y 649.136,Z 653.5,A -85,B 0,C 180,E1 31291.768,E2 31291.768} C_VEL
LIN {X 0,Y 648.771,Z 651.855,A -85,B 0,C 180,E1 31291.409,E2 31291.409} C_VEL
LIN {X 0,Y 648.768,Z 651.859,A -85,B 0,C 180,E1 31288.19,E2 31288.19} C_VEL
LIN {X 0,Y 648.764,Z 651.856,A -85,B 0,C 180,E1 31285.017,E2 31285.017} C_VEL
LIN {X 0,Y 648.76,Z 651.86,A -85,B 0,C 180,E1 31281.827,E2 31281.827} C_VEL
LIN {X 0,Y 648.772,Z 652.018,A -85,B 0,C 180,E1 31279.504,E2 31279.504} C_VEL
LIN {X 0,Y 650.145,Z 655.44,A -85,B 0,C 180,E1 31278.834,E2 31278.834} C_VEL
LIN {X 0,Y 651.64,Z 657.55,A -85,B 0,C 180,E1 31278.363,E2 31278.363} C_VEL
LIN {X 0,Y 653.571,Z 661.298,A -85,B 0,C 180,E1 31277.689,E2 31277.689} C_VEL
LIN {X 0,Y 656.823,Z 668.071,A -85,B 0,C 180,E1 31276.641,E2 31276.641} C_VEL
LIN {X 0,Y 661.072,Z 677.054,A -85,B 0,C 180,E1 31275.427,E2 31275.427} C_VEL
LIN {X 0,Y 665.167,Z 687.183,A -85,B 0,C 180,E1 31274.273,E2 31274.273} C_VEL
LIN {X 0,Y 661.497,Z 728.79,A -85,B 0,C 180,E1 31271.744,E2 31271.744} C_VEL
LIN {X 0,Y 659.099,Z 773.842,A -85,B 0,C 180,E1 31269.129,E2 31269.129} C_VEL
LIN {X 0,Y 660.155,Z 794.021,A -85,B 0,C 180,E1 31267.896,E2 31267.896} C_VEL
LIN {X 0,Y 662.836,Z 809.372,A -85,B 0,C 180,E1 31266.895,E2 31266.895} C_VEL
LIN {X 0,Y 666.997,Z 822.376,A -85,B 0,C 180,E1 31265.988,E2 31265.988} C_VEL
LIN {X 0,Y 672.825,Z 834.127,A -85,B 0,C 180,E1 31265.106,E2 31265.106} C_VEL
LIN {X 0,Y 680.541,Z 844.773,A -85,B 0,C 180,E1 31264.242,E2 31264.242} C_VEL
LIN {X 0,Y 689.33,Z 853.433,A -85,B 0,C 180,E1 31263.482,E2 31263.482} C_VEL
LIN {X 0,Y 699.32,Z 860.631,A -85,B 0,C 180,E1 31262.783,E2 31262.783} C_VEL
LIN {X 0,Y 710.793,Z 866.54,A -85,B 0,C 180,E1 31262.121,E2 31262.121} C_VEL
LIN {X 0,Y 719.138,Z 869.543,A -85,B 0,C 180,E1 31261.687,E2 31261.687} C_VEL
LIN {X 0,Y 723.621,Z 870.253,A -85,B 0,C 180,E1 31261.356,E2 31261.356} C_VEL
LIN {X 0,Y 727.616,Z 869.896,A -85,B 0,C 180,E1 31260.926,E2 31260.926} C_VEL
LIN {X 0,Y 730.037,Z 868.693,A -85,B 0,C 180,E1 31260.513,E2 31260.513} C_VEL
LIN {X 0,Y 730.434,Z 868.34,A -85,B 0,C 180,E1 31260.412,E2 31260.412} C_VEL
LIN {X 0,Y 725.051,Z 884.094,A -85,B 0,C 180,E1 31260.129,E2 31260.129} C_VEL
LIN {X 0,Y 723.542,Z 888.069,A -85,B 0,C 180,E1 31260.067,E2 31260.067} C_VEL
LIN {X 0,Y 715.192,Z 905.2,A -85,B 0,C 180,E1 31259.91,E2 31259.91} C_VEL
LIN {X 0,Y 705.412,Z 921.772,A -85,B 0,C 180,E1 31259.648,E2 31259.648} C_VEL
LIN {X 0,Y 692.792,Z 940.617,A -85,B 0,C 180,E1 31259.169,E2 31259.169} C_VEL
LIN {X 0,Y 681.087,Z 959.579,A -85,B 0,C 180,E1 31258.592,E2 31258.592} C_VEL
LIN {X 0,Y 673.618,Z 974.705,A -85,B 0,C 180,E1 31258.068,E2 31258.068} C_VEL
LIN {X 0,Y 669.509,Z 985.096,A -85,B 0,C 180,E1 31257.674,E2 31257.674} C_VEL
LIN {X 0,Y 663.851,Z 997.865,A -85,B 0,C 180,E1 31257.2,E2 31257.2} C_VEL
LIN {X 0,Y 657.67,Z 1018.349,A -85,B 0,C 180,E1 31256.354,E2 31256.354} C_VEL
LIN {X 0,Y 656.884,Z 1022.192,A -85,B 0,C 180,E1 31256.213,E2 31256.213} C_VEL
LIN {X 0,Y 656.441,Z 1063.475,A -85,B 0,C 180,E1 31255.725,E2 31255.725} C_VEL
LIN {X 0,Y 655.937,Z 1087.225,A -85,B 0,C 180,E1 31255.276,E2 31255.276} C_VEL
LIN {X 0,Y 655.368,Z 1109.696,A -85,B 0,C 180,E1 31254.685,E2 31254.685} C_VEL
LIN {X 0,Y 654.666,Z 1131.376,A -85,B 0,C 180,E1 31253.944,E2 31253.944} C_VEL
LIN {X 0,Y 653.901,Z 1152.662,A -85,B 0,C 180,E1 31253.043,E2 31253.043} C_VEL
LIN {X 0,Y 653.067,Z 1173.428,A -85,B 0,C 180,E1 31251.982,E2 31251.982} C_VEL
LIN {X 0,Y 652.297,Z 1191.367,A -85,B 0,C 180,E1 31250.895,E2 31250.895} C_VEL
LIN {X 0,Y 651.557,Z 1205.985,A -85,B 0,C 180,E1 31249.823,E2 31249.823} C_VEL
LIN {X 0,Y 650.85,Z 1219.613,A -85,B 0,C 180,E1 31248.68,E2 31248.68} C_VEL
LIN {X 0,Y 650.16,Z 1233.516,A -85,B 0,C 180,E1 31247.357,E2 31247.357} C_VEL
LIN {X 0,Y 649.471,Z 1248.326,A -85,B 0,C 180,E1 31245.72,E2 31245.72} C_VEL
LIN {X 0,Y 648.972,Z 1260.23,A -85,B 0,C 180,E1 31244.179,E2 31244.179} C_VEL
LIN {X 0,Y 648.597,Z 1270.682,A -85,B 0,C 180,E1 31242.617,E2 31242.617} C_VEL
LIN {X 0,Y 648.269,Z 1281.599,A -85,B 0,C 180,E1 31240.665,E2 31240.665} C_VEL
LIN {X 0,Y 648.092,Z 1289.367,A -85,B 0,C 180,E1 31238.963,E2 31238.963} C_VEL
LIN {X 0,Y 647.989,Z 1296.049,A -85,B 0,C 180,E1 31237.162,E2 31237.162} C_VEL
LIN {X 0,Y 647.933,Z 1301.601,A -85,B 0,C 180,E1 31235.134,E2 31235.134} C_VEL
LIN {X 0,Y 647.919,Z 1304.805,A -85,B 0,C 180,E1 31233.449,E2 31233.449} C_VEL
LIN {X 0,Y 647.907,Z 1306.918,A -85,B 0,C 180,E1 31231.591,E2 31231.591} C_VEL
LIN {X 0,Y 647.9,Z 1307.387,A -85,B 0,C 180,E1 31229.557,E2 31229.557} C_VEL
LIN {X 0,Y 647.908,Z 1306.43,A -85,B 0,C 180,E1 31227.876,E2 31227.876} C_VEL
LIN {X 0,Y 647.911,Z 1304.107,A -85,B 0,C 180,E1 31226.105,E2 31226.105} C_VEL
LIN {X 0,Y 647.935,Z 1299.636,A -85,B 0,C 180,E1 31224.064,E2 31224.064} C_VEL
LIN {X 0,Y 648.005,Z 1294.437,A -85,B 0,C 180,E1 31222.373,E2 31222.373} C_VEL
LIN {X 0,Y 648.128,Z 1287.861,A -85,B 0,C 180,E1 31220.677,E2 31220.677} C_VEL
LIN {X 0,Y 648.354,Z 1278.333,A -85,B 0,C 180,E1 31218.704,E2 31218.704} C_VEL
LIN {X 0,Y 648.65,Z 1268.77,A -85,B 0,C 180,E1 31217.083,E2 31217.083} C_VEL
LIN {X 0,Y 649.027,Z 1258.907,A -85,B 0,C 180,E1 31215.638,E2 31215.638} C_VEL
LIN {X 0,Y 649.615,Z 1245.275,A -85,B 0,C 180,E1 31213.914,E2 31213.914} C_VEL
LIN {X 0,Y 650.248,Z 1231.442,A -85,B 0,C 180,E1 31212.437,E2 31212.437} C_VEL
LIN {X 0,Y 650.905,Z 1218.56,A -85,B 0,C 180,E1 31211.226,E2 31211.226} C_VEL
LIN {X 0,Y 651.751,Z 1202.512,A -85,B 0,C 180,E1 31209.9,E2 31209.9} C_VEL
LIN {X 0,Y 652.52,Z 1186.646,A -85,B 0,C 180,E1 31208.798,E2 31208.798} C_VEL
LIN {X 0,Y 653.372,Z 1167.303,A -85,B 0,C 180,E1 31207.661,E2 31207.661} C_VEL
LIN {X 0,Y 654.228,Z 1146.367,A -85,B 0,C 180,E1 31206.633,E2 31206.633} C_VEL
LIN {X 0,Y 655.052,Z 1124.599,A -85,B 0,C 180,E1 31205.756,E2 31205.756} C_VEL
LIN {X 0,Y 655.786,Z 1102.382,A -85,B 0,C 180,E1 31205.04,E2 31205.04} C_VEL
LIN {X 0,Y 656.397,Z 1079.75,A -85,B 0,C 180,E1 31204.491,E2 31204.491} C_VEL
LIN {X 0,Y 656.838,Z 1056.743,A -85,B 0,C 180,E1 31204.103,E2 31204.103} C_VEL
LIN {X 0,Y 657.357,Z 1021.646,A -85,B 0,C 180,E1 31203.679,E2 31203.679} C_VEL
LIN {X 0,Y 660.827,Z 1009.137,A -85,B 0,C 180,E1 31203.149,E2 31203.149} C_VEL
LIN {X 0,Y 665.541,Z 995.001,A -85,B 0,C 180,E1 31202.581,E2 31202.581} C_VEL
LIN {X 0,Y 671.351,Z 981.993,A -85,B 0,C 180,E1 31202.117,E2 31202.117} C_VEL
LIN {X 0,Y 676.787,Z 968.79,A -85,B 0,C 180,E1 31201.641,E2 31201.641} C_VEL
LIN {X 0,Y 685.586,Z 952.462,A -85,B 0,C 180,E1 31201.134,E2 31201.134} C_VEL
LIN {X 0,Y 700.786,Z 928.861,A -85,B 0,C 180,E1 31200.511,E2 31200.511} C_VEL
LIN {X 0,Y 711.012,Z 912.614,A -85,B 0,C 180,E1 31200.191,E2 31200.191} C_VEL
LIN {X 0,Y 719.838,Z 896.141,A -85,B 0,C 180,E1 31199.996,E2 31199.996} C_VEL
LIN {X 0,Y 724.649,Z 885.299,A -85,B 0,C 180,E1 31199.901,E2 31199.901} C_VEL
LIN {X 0,Y 729.621,Z 870.766,A -85,B 0,C 180,E1 31199.622,E2 31199.622} C_VEL
LIN {X 0,Y 730.447,Z 868.294,A -85,B 0,C 180,E1 31199.587,E2 31199.587} C_VEL
LIN {X 0,Y 728.046,Z 869.767,A -85,B 0,C 180,E1 31199.134,E2 31199.134} C_VEL
LIN {X 0,Y 724.31,Z 870.275,A -85,B 0,C 180,E1 31198.706,E2 31198.706} C_VEL
LIN {X 0,Y 719.925,Z 869.729,A -85,B 0,C 180,E1 31198.363,E2 31198.363} C_VEL
LIN {X 0,Y 708.608,Z 865.812,A -85,B 0,C 180,E1 31197.697,E2 31197.697} C_VEL
